KUKA KRL program: MyProgram_042().src

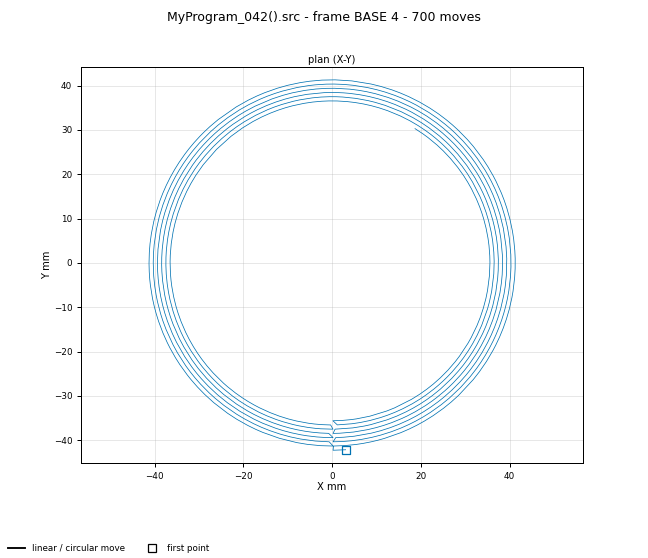
[picture p0: tool path of MyProgram_042().src in frame BASE 4, 700 of 700 moves have a stored position in this frame; points joined in program order, loops and branches not executed]
&ACCESS RVP
&REL 1
&PARAM TEMPLATE = C:\KRC\Roboter\Template\vorgabe
&PARAM EDITMASK = *
DEF MyProgram_042()
; ---- Setting reference (Base) ----
$BASE = BASE_DATA[4]

; --------------------------
; ---- Setting tool (TCP) ----
$TOOL = TOOL_DATA[3]
; --------------------------

$VEL.CP = VEL_APROX_PRINT
Startdeposition()
$VEL.CP = VEL_PRINT
LIN {X 3.0442,Y -42.1231,Z 63,A -93.24,B 24.8701,C -2.6301,E1 25.0087,E2 -183.3555} C_DIS
LIN {X 0.2102,Y -42.232,Z 63,A -95.217,B 24.8675,C -2.6563,E1 25.0033,E2 -181.4412} C_DIS
Enddeposition()
LIN {X 0.2102,Y -42.232,Z 63,A -95.217,B 24.8675,C -2.6563,E1 25.0033,E2 -181.4412} C_DIS
Startdeposition()
$VEL.CP = VEL_PRINT
LIN {X 0.315,Y -41.2814,Z 63,A -95.2944,B 24.8662,C -2.6692,E1 25.0033,E2 -181.3947} C_DIS
LIN {X 2.8307,Y -41.1855,Z 63,A -91.2878,B 24.8653,C -2.6781,E1 25.0144,E2 -185.421} C_DIS
LIN {X 5.3557,Y -40.9338,Z 63,A -88.2842,B 24.8659,C -2.6725,E1 25.0227,E2 -188.409} C_DIS
LIN {X 6.9926,Y -40.6865,Z 63,A -85.9418,B 24.8656,C -2.6748,E1 25.0292,E2 -190.7546} C_DIS
LIN {X 8.7788,Y -40.3384,Z 63,A -83.5592,B 24.8656,C -2.6748,E1 25.0357,E2 -193.1343} C_DIS
LIN {X 10.339,Y -39.9671,Z 63,A -81.3025,B 24.8654,C -2.6775,E1 25.0418,E2 -195.3939} C_DIS
LIN {X 11.8031,Y -39.5594,Z 63,A -78.4268,B 24.8639,C -2.6916,E1 25.0496,E2 -198.2983} C_DIS
LIN {X 15.4835,Y -38.2691,Z 63,A -73.5141,B 24.864,C -2.6909,E1 25.0624,E2 -203.1988} C_DIS
LIN {X 17.356,Y -37.457,Z 63,A -70.9592,B 24.864,C -2.6907,E1 25.0689,E2 -205.747} C_DIS
LIN {X 19.1269,Y -36.5846,Z 63,A -67.9342,B 24.8631,C -2.6997,E1 25.0765,E2 -208.785} C_DIS
LIN {X 20.771,Y -35.6773,Z 63,A -65.7267,B 24.8633,C -2.6979,E1 25.0818,E2 -210.9816} C_DIS
LIN {X 22.743,Y -34.453,Z 63,A -61.7056,B 24.8614,C -2.7169,E1 25.0913,E2 -215.0347} C_DIS
LIN {X 25.1016,Y -32.7747,Z 63,A -58.6078,B 24.8621,C -2.7101,E1 25.0982,E2 -218.1053} C_DIS
LIN {X 26.8177,Y -31.3859,Z 63,A -54.5171,B 24.8596,C -2.7337,E1 25.1071,E2 -222.2362} C_DIS
LIN {X 28.5068,Y -29.8606,Z 63,A -51.198,B 24.8586,C -2.7437,E1 25.1138,E2 -225.5653} C_DIS
LIN {X 31.826,Y -26.2941,Z 63,A -45.9801,B 24.8596,C -2.7345,E1 25.1235,E2 -230.7384} C_DIS
LIN {X 33.2022,Y -24.5336,Z 63,A -41.6673,B 24.8566,C -2.7631,E1 25.1308,E2 -235.0984} C_DIS
LIN {X 34.8038,Y -22.2027,Z 63,A -38.0776,B 24.8561,C -2.7682,E1 25.1363,E2 -238.682} C_DIS
LIN {X 36.2645,Y -19.7265,Z 63,A -34.6826,B 24.856,C -2.7693,E1 25.141,E2 -242.0622} C_DIS
LIN {X 36.8871,Y -18.5378,Z 63,A -32.5636,B 24.8549,C -2.7791,E1 25.1437,E2 -244.193} C_DIS
LIN {X 37.7579,Y -16.6921,Z 63,A -29.815,B 24.8542,C -2.786,E1 25.1469,E2 -246.9431} C_DIS
LIN {X 38.5649,Y -14.7316,Z 63,A -26.6228,B 24.8528,C -2.7991,E1 25.1502,E2 -250.1487} C_DIS
LIN {X 39.282,Y -12.6955,Z 63,A -23.7097,B 24.852,C -2.8068,E1 25.1528,E2 -253.0635} C_DIS
LIN {X 39.9316,Y -10.477,Z 63,A -20.4876,B 24.8509,C -2.8169,E1 25.1552,E2 -256.291} C_DIS
LIN {X 40.5343,Y -7.8247,Z 63,A -17.1592,B 24.8505,C -2.8209,E1 25.1571,E2 -259.6096} C_DIS
LIN {X 40.7866,Y -6.3807,Z 63,A -14.5033,B 24.8487,C -2.8381,E1 25.1583,E2 -262.2905} C_DIS
LIN {X 41.1553,Y -3.24,Z 63,A -10.513,B 24.8479,C -2.8449,E1 25.1594,E2 -266.2733} C_DIS
LIN {X 41.2627,Y -1.282,Z 63,A -7.9389,B 24.8473,C -2.8509,E1 25.1597,E2 -268.8463} C_DIS
LIN {X 41.2709,Y 1.0166,Z 63,A -4.6576,B 24.8461,C -2.8625,E1 25.1597,E2 -272.1355} C_DIS
LIN {X 41.1906,Y 2.7556,Z 63,A -2.0891,B 24.845,C -2.8727,E1 25.1592,E2 -274.7128} C_DIS
LIN {X 40.9304,Y 5.3819,Z 63,A 1.2618,B 24.8443,C -2.8786,E1 25.1582,E2 -278.0579} C_DIS
LIN {X 40.6503,Y 7.1984,Z 63,A 3.8015,B 24.8435,C -2.8862,E1 25.157,E2 -280.6007} C_DIS
LIN {X 40.085,Y 9.8718,Z 63,A 7.7678,B 24.8419,C -2.9006,E1 25.1546,E2 -284.5781} C_DIS
LIN {X 39.3831,Y 12.3781,Z 63,A 11.2245,B 24.841,C -2.9086,E1 25.1519,E2 -288.0339} C_DIS
LIN {X 38.8049,Y 14.0869,Z 63,A 13.9911,B 24.8397,C -2.9203,E1 25.1493,E2 -290.8127} C_DIS
LIN {X 38.1479,Y 15.7808,Z 63,A 16.574,B 24.8388,C -2.9285,E1 25.1465,E2 -293.4007} C_DIS
LIN {X 36.9226,Y 18.4657,Z 63,A 20.0406,B 24.8388,C -2.9291,E1 25.1424,E2 -296.85} C_DIS
LIN {X 36.2981,Y 19.6648,Z 63,A 22.4905,B 24.8372,C -2.9437,E1 25.1392,E2 -299.3218} C_DIS
LIN {X 35.1309,Y 21.6821,Z 63,A 25.3607,B 24.8369,C -2.946,E1 25.1351,E2 -302.1826} C_DIS
LIN {X 34.0764,Y 23.3033,Z 63,A 28.3406,B 24.8356,C -2.9576,E1 25.1304,E2 -305.1752} C_DIS
LIN {X 31.8607,Y 26.2512,Z 63,A 33.4994,B 24.8342,C -2.9703,E1 25.1215,E2 -310.3398} C_DIS
LIN {X 30.509,Y 27.8114,Z 63,A 36.4108,B 24.8334,C -2.9773,E1 25.1161,E2 -313.2549} C_DIS
LIN {X 28.3817,Y 29.9792,Z 63,A 40.0226,B 24.8335,C -2.9762,E1 25.1089,E2 -316.8489} C_DIS
LIN {X 27.0729,Y 31.1661,Z 63,A 42.6358,B 24.8327,C -2.9835,E1 25.1035,E2 -319.469} C_DIS
LIN {X 25.7131,Y 32.2973,Z 63,A 45.1305,B 24.8321,C -2.9886,E1 25.0981,E2 -321.9664} C_DIS
LIN {X 23.9669,Y 33.6129,Z 63,A 48.357,B 24.8312,C -2.9968,E1 25.0908,E2 -325.2008} C_DIS
LIN {X 22.0438,Y 34.9044,Z 63,A 51.6022,B 24.8306,C -3.0022,E1 25.0832,E2 -328.4482} C_DIS
LIN {X 19.7088,Y 36.2742,Z 63,A 55.2508,B 24.8302,C -3.0056,E1 25.0743,E2 -332.0942} C_DIS
LIN {X 17.2496,Y 37.5061,Z 63,A 58.8402,B 24.8301,C -3.0067,E1 25.0653,E2 -335.6767} C_DIS
LIN {X 15.2686,Y 38.3557,Z 63,A 61.9376,B 24.8296,C -3.0113,E1 25.0573,E2 -338.7779} C_DIS
LIN {X 13.4538,Y 39.0293,Z 63,A 64.4175,B 24.8296,C -3.0106,E1 25.0508,E2 -341.2509} C_DIS
LIN {X 11.0382,Y 39.7796,Z 63,A 68.6726,B 24.8281,C -3.024,E1 25.0393,E2 -345.5307} C_DIS
LIN {X 8.7687,Y 40.3406,Z 63,A 72.0577,B 24.8277,C -3.0276,E1 25.0301,E2 -348.9199} C_DIS
LIN {X 4.4531,Y 41.042,Z 63,A 77.9984,B 24.8277,C -3.0271,E1 25.0137,E2 -354.8545} C_DIS
LIN {X 0.6654,Y 41.2774,Z 63,A 82.6151,B 24.8288,C -3.0177,E1 25.0008,E2 -359.4473} C_DIS
LIN {X -2.2833,Y 41.2194,Z 63,A 87.1591,B 24.8283,C -3.0226,E1 24.9881,E2 -364.0039} C_DIS
LIN {X -5.0199,Y 40.9768,Z 63,A 90.6583,B 24.829,C -3.0164,E1 24.9784,E2 -367.4903} C_DIS
LIN {X -7.1609,Y 40.6571,Z 63,A 93.4772,B 24.8295,C -3.0118,E1 24.9707,E2 -370.3009} C_DIS
LIN {X -9.9422,Y 40.0677,Z 63,A 98.312,B 24.8286,C -3.02,E1 24.9575,E2 -375.1616} C_DIS
LIN {X -12.3271,Y 39.3993,Z 63,A 101.3903,B 24.8295,C -3.0115,E1 24.9493,E2 -378.225} C_DIS
LIN {X -15.2193,Y 38.3746,Z 63,A 105.1565,B 24.8309,C -2.9998,E1 24.9395,E2 -381.971} C_DIS
LIN {X -16.9866,Y 37.6259,Z 63,A 107.9518,B 24.8311,C -2.9977,E1 24.9324,E2 -384.7678} C_DIS
LIN {X -18.9393,Y 36.6822,Z 63,A 111.1263,B 24.8314,C -2.995,E1 24.9244,E2 -387.9443} C_DIS
LIN {X -21.6363,Y 35.1594,Z 63,A 116.2699,B 24.8311,C -2.9978,E1 24.912,E2 -393.1102} C_DIS
LIN {X -25.6799,Y 32.3235,Z 63,A 122.2724,B 24.8338,C -2.9736,E1 24.8986,E2 -399.0763} C_DIS
LIN {X -27.5314,Y 30.7617,Z 63,A 125.6343,B 24.8346,C -2.9662,E1 24.8916,E2 -402.4337} C_DIS
LIN {X -28.875,Y 29.5046,Z 63,A 127.9005,B 24.8357,C -2.957,E1 24.887,E2 -404.6872} C_DIS
LIN {X -29.8566,Y 28.5109,Z 63,A 129.8633,B 24.8362,C -2.9526,E1 24.8832,E2 -406.648} C_DIS
LIN {X -31.0997,Y 27.1489,Z 63,A 132.6919,B 24.8365,C -2.9494,E1 24.8779,E2 -409.4817} C_DIS
LIN {X -32.2803,Y 25.7346,Z 63,A 134.9712,B 24.8376,C -2.9397,E1 24.8739,E2 -411.7483} C_DIS
LIN {X -33.2684,Y 24.4433,Z 63,A 137.2968,B 24.8382,C -2.9346,E1 24.87,E2 -414.0728} C_DIS
LIN {X -34.5023,Y 22.6682,Z 63,A 140.7751,B 24.8385,C -2.9319,E1 24.8646,E2 -417.5619} C_DIS
LIN {X -35.5264,Y 21.0269,Z 63,A 143.1596,B 24.8397,C -2.921,E1 24.8612,E2 -419.9327} C_DIS
LIN {X -36.4931,Y 19.3006,Z 63,A 145.7888,B 24.8407,C -2.9119,E1 24.8577,E2 -422.5541} C_DIS
LIN {X -37.4028,Y 17.4725,Z 63,A 148.9048,B 24.8412,C -2.9068,E1 24.8539,E2 -425.6746} C_DIS
LIN {X -38.1649,Y 15.7395,Z 63,A 151.2341,B 24.8424,C -2.8957,E1 24.8514,E2 -427.9904} C_DIS
LIN {X -38.7933,Y 14.1186,Z 63,A 153.8854,B 24.8429,C -2.8911,E1 24.8488,E2 -430.6456} C_DIS
LIN {X -39.6647,Y 11.4457,Z 63,A 157.3648,B 24.8447,C -2.8746,E1 24.8459,E2 -434.1055} C_DIS
LIN {X -40.2119,Y 9.3412,Z 63,A 161.2523,B 24.8447,C -2.8748,E1 24.8432,E2 -438.0161} C_DIS
LIN {X -40.7666,Y 6.5072,Z 63,A 165.1234,B 24.8462,C -2.8608,E1 24.8414,E2 -441.8767} C_DIS
LIN {X -41.0514,Y 4.3638,Z 63,A 167.693,B 24.8478,C -2.8467,E1 24.8405,E2 -444.4279} C_DIS
LIN {X -41.2148,Y 2.3664,Z 63,A 170.8387,B 24.8483,C -2.8419,E1 24.8399,E2 -447.5811} C_DIS
LIN {X -41.2825,Y -0.1257,Z 63,A 173.8276,B 24.85,C -2.826,E1 24.8398,E2 -450.5498} C_DIS
LIN {X -41.2319,Y -2.0447,Z 63,A 176.7215,B 24.8506,C -2.8201,E1 24.8401,E2 -453.4472} C_DIS
LIN {X -41.1157,Y -3.7096,Z 63,A 178.9624,B 24.8514,C -2.8121,E1 24.8406,E2 -455.6824} C_DIS
LIN {X -40.9765,Y -5.0234,Z 63,A -178.6298,B 24.8514,C -2.8128,E1 24.8414,E2 -458.1061} C_DIS
LIN {X -40.4873,Y -8.0658,Z 63,A -174.7424,B 24.8532,C -2.7954,E1 24.8432,E2 -461.9751} C_DIS
LIN {X -40.0866,Y -9.8654,Z 63,A -172.1473,B 24.854,C -2.7882,E1 24.8449,E2 -464.568} C_DIS
LIN {X -39.674,Y -11.413,Z 63,A -170.0611,B 24.8548,C -2.7801,E1 24.8464,E2 -466.6469} C_DIS
LIN {X -39.1144,Y -13.2029,Z 63,A -167.1196,B 24.8552,C -2.7763,E1 24.849,E2 -469.5962} C_DIS
LIN {X -38.1488,Y -15.7789,Z 63,A -163.1877,B 24.8562,C -2.7667,E1 24.853,E2 -473.5272} C_DIS
LIN {X -37.1675,Y -17.9678,Z 63,A -160.3099,B 24.8577,C -2.7524,E1 24.8564,E2 -476.3866} C_DIS
LIN {X -36.5638,Y -19.1664,Z 63,A -158.0107,B 24.8577,C -2.7524,E1 24.8593,E2 -478.6981} C_DIS
LIN {X -35.3355,Y -21.3457,Z 63,A -154.537,B 24.8586,C -2.7434,E1 24.8642,E2 -482.1684} C_DIS
LIN {X -34.341,Y -22.9129,Z 63,A -151.7472,B 24.859,C -2.7395,E1 24.8685,E2 -484.9627} C_DIS
LIN {X -32.6576,Y -25.2536,Z 63,A -148.3403,B 24.8607,C -2.723,E1 24.8741,E2 -488.3465} C_DIS
LIN {X -31.8669,Y -26.2441,Z 63,A -146.1604,B 24.8607,C -2.7239,E1 24.878,E2 -490.5388} C_DIS
LIN {X -30.3612,Y -27.9725,Z 63,A -143.0206,B 24.8614,C -2.7164,E1 24.8838,E2 -493.6748} C_DIS
LIN {X -28.7127,Y -29.6617,Z 63,A -139.6987,B 24.862,C -2.7103,E1 24.8904,E2 -496.996} C_DIS
LIN {X -26.6654,Y -31.5156,Z 63,A -135.2889,B 24.862,C -2.7101,E1 24.8997,E2 -501.4227} C_DIS
LIN {X -23.5731,Y -33.8905,Z 63,A -130.0918,B 24.8633,C -2.6983,E1 24.9114,E2 -506.6101} C_DIS
LIN {X -21.5024,Y -35.2407,Z 63,A -126.7529,B 24.8639,C -2.6921,E1 24.9193,E2 -509.9447} C_DIS
LIN {X -19.0548,Y -36.6218,Z 63,A -123.185,B 24.8648,C -2.6828,E1 24.928,E2 -513.5004} C_DIS
LIN {X -17.1898,Y -37.5339,Z 63,A -120.338,B 24.8652,C -2.679,E1 24.9352,E2 -516.3457} C_DIS
LIN {X -15.6398,Y -38.2055,Z 63,A -117.3395,B 24.8646,C -2.6854,E1 24.943,E2 -519.3661} C_DIS
LIN {X -11.9039,Y -39.5295,Z 63,A -111.6303,B 24.8647,C -2.684,E1 24.9581,E2 -525.0825} C_DIS
LIN {X -7.9714,Y -40.5061,Z 63,A -107.0486,B 24.8664,C -2.6669,E1 24.9705,E2 -529.6295} C_DIS
LIN {X -5.6211,Y -40.8983,Z 63,A -102.6413,B 24.865,C -2.6816,E1 24.9828,E2 -534.0754} C_DIS
LIN {X -2.6104,Y -41.2002,Z 63,A -98.9251,B 24.8657,C -2.6746,E1 24.9931,E2 -537.7766} C_DIS
LIN {X 0.2191,Y -41.2805,Z 63,A -96.8151,B 24.8682,C -2.6493,E1 24.9988,E2 -539.8267} C_DIS
Enddeposition()
LIN {X 0.2191,Y -41.2805,Z 63,A -96.8151,B 24.8682,C -2.6493,E1 24.9988,E2 -539.8267} C_DIS
Startdeposition()
$VEL.CP = VEL_PRINT
LIN {X -0.6723,Y -40.3269,Z 63,A -98.638,B 24.8673,C -2.6582,E1 24.9938,E2 -538.0247} C_DIS
LIN {X -3.7987,Y -40.1536,Z 63,A -102.8793,B 24.867,C -2.661,E1 24.982,E2 -533.7884} C_DIS
LIN {X -7.1068,Y -39.7017,Z 63,A -106.8696,B 24.8659,C -2.6722,E1 24.971,E2 -529.8212} C_DIS
LIN {X -9.4207,Y -39.2174,Z 63,A -111.0995,B 24.8669,C -2.6624,E1 24.9594,E2 -525.5625} C_DIS
LIN {X -11.7387,Y -38.5874,Z 63,A -114.2382,B 24.8663,C -2.6681,E1 24.9511,E2 -522.4324} C_DIS
LIN {X -14.0146,Y -37.82,Z 63,A -117.3497,B 24.8657,C -2.6747,E1 24.9429,E2 -519.3306} C_DIS
LIN {X -15.9354,Y -37.0518,Z 63,A -120.4596,B 24.8656,C -2.6755,E1 24.9348,E2 -516.2155} C_DIS
LIN {X -17.6856,Y -36.2491,Z 63,A -122.93,B 24.8649,C -2.6819,E1 24.9286,E2 -513.754} C_DIS
LIN {X -19.7095,Y -35.1891,Z 63,A -126.7906,B 24.8653,C -2.6786,E1 24.9191,E2 -509.8748} C_DIS
LIN {X -21.525,Y -34.1093,Z 63,A -129.8482,B 24.8649,C -2.6824,E1 24.9119,E2 -506.8163} C_DIS
LIN {X -24.3338,Y -32.1655,Z 63,A -134.5954,B 24.8639,C -2.6916,E1 24.9011,E2 -502.0747} C_DIS
LIN {X -26.3607,Y -30.5267,Z 63,A -138.0135,B 24.8629,C -2.7017,E1 24.8938,E2 -498.6676} C_DIS
LIN {X -27.723,Y -29.2947,Z 63,A -140.8695,B 24.8627,C -2.7041,E1 24.888,E2 -495.8055} C_DIS
LIN {X -29.6846,Y -27.305,Z 63,A -144.4563,B 24.8614,C -2.7168,E1 24.8811,E2 -492.2336} C_DIS
LIN {X -30.9078,Y -25.9128,Z 63,A -147.0794,B 24.8608,C -2.7227,E1 24.8763,E2 -489.6128} C_DIS
LIN {X -31.9763,Y -24.5815,Z 63,A -149.52,B 24.8602,C -2.7282,E1 24.8721,E2 -487.1738} C_DIS
LIN {X -32.9916,Y -23.2011,Z 63,A -152.5473,B 24.8602,C -2.7276,E1 24.8672,E2 -484.1302} C_DIS
LIN {X -34.8756,Y -20.2598,Z 63,A -157.4876,B 24.8589,C -2.7405,E1 24.86,E2 -479.1955} C_DIS
LIN {X -35.8631,Y -18.4549,Z 63,A -160.6337,B 24.8584,C -2.746,E1 24.8559,E2 -476.0457} C_DIS
LIN {X -37.4233,Y -15.0421,Z 63,A -165.3478,B 24.8562,C -2.7673,E1 24.8507,E2 -471.3567} C_DIS
LIN {X -38.1586,Y -13.0647,Z 63,A -168.5623,B 24.8555,C -2.7737,E1 24.8477,E2 -468.1391} C_DIS
LIN {X -38.6645,Y -11.48,Z 63,A -171.1673,B 24.855,C -2.7781,E1 24.8456,E2 -465.5297} C_DIS
LIN {X -39.3705,Y -8.7591,Z 63,A -174.6366,B 24.8532,C -2.7955,E1 24.8433,E2 -462.0816} C_DIS
LIN {X -39.6731,Y -7.2657,Z 63,A -177.011,B 24.8527,C -2.7999,E1 24.8421,E2 -459.7037} C_DIS
LIN {X -39.9923,Y -5.2302,Z 63,A -179.865,B 24.8517,C -2.8096,E1 24.8409,E2 -456.856} C_DIS
LIN {X -40.2241,Y -2.9686,Z 63,A 176.0361,B 24.8516,C -2.8108,E1 24.84,E2 -452.7352} C_DIS
LIN {X -40.3332,Y 0.0142,Z 63,A 172.5148,B 24.8494,C -2.8313,E1 24.8398,E2 -449.2418} C_DIS
LIN {X -40.279,Y 2.0829,Z 63,A 169.4008,B 24.8486,C -2.8388,E1 24.8401,E2 -446.1269} C_DIS
LIN {X -40.1128,Y 4.2063,Z 63,A 165.9993,B 24.848,C -2.8445,E1 24.8411,E2 -442.7187} C_DIS
LIN {X -39.6244,Y 7.5267,Z 63,A 161.4804,B 24.8461,C -2.8618,E1 24.8431,E2 -438.2145} C_DIS
LIN {X -38.9796,Y 10.3609,Z 63,A 157.4198,B 24.8447,C -2.8753,E1 24.8458,E2 -434.1624} C_DIS
LIN {X -38.1564,Y 13.0713,Z 63,A 153.0309,B 24.8437,C -2.8838,E1 24.8496,E2 -429.7687} C_DIS
LIN {X -37.1679,Y 15.6614,Z 63,A 149.2433,B 24.8423,C -2.8971,E1 24.8535,E2 -425.9918} C_DIS
LIN {X -36.2263,Y 17.7322,Z 63,A 146.4377,B 24.8408,C -2.9109,E1 24.8569,E2 -423.204} C_DIS
LIN {X -35.3698,Y 19.384,Z 63,A 143.596,B 24.8402,C -2.9164,E1 24.8606,E2 -420.3603} C_DIS
LIN {X -34.4492,Y 20.9759,Z 63,A 141.2131,B 24.8391,C -2.9261,E1 24.864,E2 -417.9884} C_DIS
LIN {X -33.4645,Y 22.5138,Z 63,A 138.3387,B 24.8387,C -2.9302,E1 24.8684,E2 -415.1093} C_DIS
LIN {X -32.4432,Y 23.9625,Z 63,A 136.0696,B 24.8376,C -2.9395,E1 24.8721,E2 -412.8515} C_DIS
LIN {X -31.4476,Y 25.255,Z 63,A 133.6511,B 24.8371,C -2.9444,E1 24.8762,E2 -410.4333} C_DIS
LIN {X -29.9352,Y 27.0299,Z 63,A 129.6912,B 24.8369,C -2.9457,E1 24.8836,E2 -406.4586} C_DIS
LIN {X -27.4236,Y 29.5748,Z 63,A 124.7893,B 24.8354,C -2.9594,E1 24.8933,E2 -401.569} C_DIS
LIN {X -25.668,Y 31.1112,Z 63,A 121.871,B 24.8341,C -2.971,E1 24.8995,E2 -398.6672} C_DIS
LIN {X -23.5027,Y 32.7775,Z 63,A 117.1805,B 24.8342,C -2.9698,E1 24.9101,E2 -393.957} C_DIS
LIN {X -20.9052,Y 34.4921,Z 63,A 113.3733,B 24.8325,C -2.9849,E1 24.919,E2 -390.1739} C_DIS
LIN {X -18.8345,Y 35.6651,Z 63,A 109.6522,B 24.8324,C -2.9866,E1 24.9281,E2 -386.4462} C_DIS
LIN {X -16.3132,Y 36.8866,Z 63,A 106.4728,B 24.8306,C -3.0021,E1 24.9361,E2 -383.2956} C_DIS
LIN {X -14.6293,Y 37.5863,Z 63,A 103.5697,B 24.8306,C -3.0018,E1 24.9436,E2 -380.3855} C_DIS
LIN {X -12.9467,Y 38.1984,Z 63,A 100.8236,B 24.8306,C -3.0025,E1 24.9509,E2 -377.6356} C_DIS
LIN {X -11.1981,Y 38.747,Z 63,A 97.7211,B 24.8309,C -2.9992,E1 24.9592,E2 -374.5202} C_DIS
LIN {X -7.9066,Y 39.5508,Z 63,A 93.2503,B 24.83,C -3.0076,E1 24.9714,E2 -370.0637} C_DIS
LIN {X -5.2768,Y 39.986,Z 63,A 89.8662,B 24.8291,C -3.0152,E1 24.9807,E2 -366.6949} C_DIS
LIN {X -3.7844,Y 40.1549,Z 63,A 87.3873,B 24.8295,C -3.0119,E1 24.9876,E2 -364.2066} C_DIS
LIN {X -1.3223,Y 40.311,Z 63,A 83.8807,B 24.8294,C -3.0131,E1 24.9973,E2 -360.7019} C_DIS
LIN {X 0.4163,Y 40.331,Z 63,A 81.3218,B 24.8294,C -3.0124,E1 25.0045,E2 -358.1415} C_DIS
LIN {X 2.6441,Y 40.2461,Z 63,A 78.4388,B 24.829,C -3.0162,E1 25.0125,E2 -355.2687} C_DIS
LIN {X 4.7439,Y 40.0529,Z 63,A 74.9846,B 24.8297,C -3.0096,E1 25.0221,E2 -351.8012} C_DIS
LIN {X 7.9549,Y 39.5409,Z 63,A 70.9226,B 24.8291,C -3.0157,E1 25.0332,E2 -347.7578} C_DIS
LIN {X 10.1713,Y 39.0292,Z 63,A 67.5872,B 24.8294,C -3.0125,E1 25.0423,E2 -344.4196} C_DIS
LIN {X 11.9463,Y 38.523,Z 63,A 64.861,B 24.8298,C -3.0091,E1 25.0496,E2 -341.6903} C_DIS
LIN {X 14.0403,Y 37.8106,Z 63,A 61.8691,B 24.8298,C -3.0086,E1 25.0575,E2 -338.703} C_DIS
LIN {X 15.6139,Y 37.1879,Z 63,A 59.3682,B 24.8303,C -3.0048,E1 25.0639,E2 -336.1988} C_DIS
LIN {X 17.4857,Y 36.3454,Z 63,A 56.573,B 24.8305,C -3.0032,E1 25.071,E2 -333.4071} C_DIS
LIN {X 19.0006,Y 35.5773,Z 63,A 53.6808,B 24.8316,C -2.9931,E1 25.0782,E2 -330.4989} C_DIS
LIN {X 21.8543,Y 33.8988,Z 63,A 49.8608,B 24.8309,C -2.9994,E1 25.0873,E2 -326.7058} C_DIS
LIN {X 23.7603,Y 32.5912,Z 63,A 45.7015,B 24.833,C -2.9808,E1 25.0968,E2 -322.5168} C_DIS
LIN {X 25.5002,Y 31.2489,Z 63,A 43.1956,B 24.8326,C -2.9846,E1 25.1023,E2 -320.0291} C_DIS
LIN {X 26.5953,Y 30.3222,Z 63,A 41.107,B 24.8331,C -2.9799,E1 25.1067,E2 -317.9377} C_DIS
LIN {X 27.705,Y 29.3117,Z 63,A 38.678,B 24.8341,C -2.9711,E1 25.1117,E2 -315.4977} C_DIS
LIN {X 29.529,Y 27.4728,Z 63,A 35.2524,B 24.8345,C -2.9673,E1 25.1183,E2 -312.0778} C_DIS
LIN {X 31.1134,Y 25.6654,Z 63,A 31.3937,B 24.8362,C -2.9526,E1 25.1253,E2 -308.2019} C_DIS
LIN {X 32.6965,Y 23.6163,Z 63,A 27.6778,B 24.8372,C -2.9432,E1 25.1315,E2 -304.4816} C_DIS
LIN {X 34.4358,Y 20.998,Z 63,A 23.9494,B 24.8372,C -2.9437,E1 25.1371,E2 -300.7731} C_DIS
LIN {X 35.1373,Y 19.8015,Z 63,A 21.9628,B 24.8378,C -2.9383,E1 25.1399,E2 -298.7839} C_DIS
LIN {X 35.8718,Y 18.4379,Z 63,A 19.7335,B 24.8385,C -2.9319,E1 25.1428,E2 -296.5513} C_DIS
LIN {X 36.7127,Y 16.7012,Z 63,A 16.6795,B 24.8399,C -2.9193,E1 25.1464,E2 -293.4839} C_DIS
LIN {X 37.4691,Y 14.9279,Z 63,A 14.2702,B 24.8401,C -2.917,E1 25.149,E2 -291.0823} C_DIS
LIN {X 38.2617,Y 12.759,Z 63,A 10.3402,B 24.8423,C -2.8969,E1 25.1526,E2 -287.1268} C_DIS
LIN {X 38.9421,Y 10.4999,Z 63,A 7.5435,B 24.8424,C -2.896,E1 25.1548,E2 -284.3442} C_DIS
LIN {X 39.5395,Y 7.9614,Z 63,A 3.4265,B 24.8444,C -2.8781,E1 25.1572,E2 -280.2087} C_DIS
LIN {X 39.942,Y 5.6015,Z 63,A -0.1327,B 24.8458,C -2.865,E1 25.1587,E2 -276.6395} C_DIS
LIN {X 40.2893,Y 1.8711,Z 63,A -4.9516,B 24.8467,C -2.8568,E1 25.1597,E2 -271.8298} C_DIS
LIN {X 40.3236,Y -0.8722,Z 63,A -9.1136,B 24.8485,C -2.8402,E1 25.1597,E2 -267.6533} C_DIS
LIN {X 40.2198,Y -3.0229,Z 63,A -12.1864,B 24.8495,C -2.8304,E1 25.1591,E2 -264.5753} C_DIS
LIN {X 39.8473,Y -6.2392,Z 63,A -16.2724,B 24.8501,C -2.8245,E1 25.1576,E2 -260.4995} C_DIS
LIN {X 39.5044,Y -8.1325,Z 63,A -18.9712,B 24.851,C -2.8165,E1 25.1561,E2 -257.7978} C_DIS
LIN {X 39.1186,Y -9.8242,Z 63,A -21.3873,B 24.8517,C -2.8097,E1 25.1546,E2 -255.3794} C_DIS
LIN {X 38.7142,Y -11.3126,Z 63,A -23.4528,B 24.8522,C -2.805,E1 25.153,E2 -253.3148} C_DIS
LIN {X 38.2315,Y -12.8487,Z 63,A -25.8167,B 24.8531,C -2.7968,E1 25.151,E2 -250.9447} C_DIS
LIN {X 37.5984,Y -14.5986,Z 63,A -28.5362,B 24.854,C -2.7876,E1 25.1483,E2 -248.2186} C_DIS
LIN {X 36.9237,Y -16.2293,Z 63,A -30.9038,B 24.8546,C -2.7824,E1 25.1457,E2 -245.8518} C_DIS
LIN {X 36.2858,Y -17.6097,Z 63,A -32.9712,B 24.8551,C -2.7776,E1 25.1432,E2 -243.7842} C_DIS
LIN {X 35.5224,Y -19.1027,Z 63,A -35.5389,B 24.8561,C -2.7677,E1 25.1399,E2 -241.2065} C_DIS
LIN {X 34.5887,Y -20.7464,Z 63,A -38.1715,B 24.8568,C -2.761,E1 25.1362,E2 -238.5716} C_DIS
LIN {X 33.5695,Y -22.3575,Z 63,A -40.9006,B 24.8576,C -2.7532,E1 25.132,E2 -235.8378} C_DIS
LIN {X 32.5771,Y -23.7795,Z 63,A -43.1766,B 24.858,C -2.7496,E1 25.1283,E2 -233.5644} C_DIS
LIN {X 31.1406,Y -25.6326,Z 63,A -46.8133,B 24.8594,C -2.736,E1 25.122,E2 -229.9125} C_DIS
LIN {X 28.9609,Y -28.0705,Z 63,A -51.7845,B 24.8611,C -2.7195,E1 25.1125,E2 -224.9239} C_DIS
LIN {X 26.4435,Y -30.4544,Z 63,A -56.8908,B 24.8625,C -2.7055,E1 25.1019,E2 -219.8049} C_DIS
LIN {X 24.6004,Y -31.9618,Z 63,A -59.5165,B 24.8621,C -2.7101,E1 25.0962,E2 -217.2} C_DIS
LIN {X 22.1544,Y -33.7034,Z 63,A -63.5632,B 24.8626,C -2.7051,E1 25.087,E2 -213.1552} C_DIS
LIN {X 20.532,Y -34.7155,Z 63,A -66.5739,B 24.8635,C -2.6956,E1 25.0797,E2 -210.1314} C_DIS
LIN {X 18.9264,Y -35.6167,Z 63,A -68.934,B 24.8636,C -2.695,E1 25.074,E2 -207.7769} C_DIS
LIN {X 17.294,Y -36.4375,Z 63,A -71.7425,B 24.8643,C -2.6877,E1 25.0669,E2 -204.9584} C_DIS
LIN {X 15.5479,Y -37.2158,Z 63,A -74.2772,B 24.8645,C -2.6865,E1 25.0604,E2 -202.4269} C_DIS
LIN {X 13.3753,Y -38.0504,Z 63,A -77.9999,B 24.8655,C -2.676,E1 25.0506,E2 -198.6872} C_DIS
LIN {X 10.9144,Y -38.828,Z 63,A -81.5928,B 24.8658,C -2.673,E1 25.041,E2 -195.0934} C_DIS
LIN {X 8.9724,Y -39.3223,Z 63,A -84.0709,B 24.8656,C -2.6756,E1 25.0343,E2 -192.6251} C_DIS
LIN {X 6.643,Y -39.782,Z 63,A -87.891,B 24.8665,C -2.6665,E1 25.0238,E2 -188.7877} C_DIS
LIN {X 4.3725,Y -40.0954,Z 63,A -90.7016,B 24.866,C -2.6708,E1 25.016,E2 -185.9895} C_DIS
LIN {X 2.215,Y -40.2719,Z 63,A -94.0044,B 24.8665,C -2.6663,E1 25.0068,E2 -182.6774} C_DIS
LIN {X 0.2157,Y -40.3237,Z 63,A -96.1344,B 24.8656,C -2.6755,E1 25.0009,E2 -180.5697} C_DIS
Enddeposition()
LIN {X 0.2157,Y -40.3237,Z 63,A -96.1344,B 24.8656,C -2.6755,E1 25.0009,E2 -180.5697} C_DIS
Startdeposition()
$VEL.CP = VEL_PRINT
LIN {X 0.8258,Y -39.3744,Z 63,A -94.5482,B 24.8629,C -2.7016,E1 25.0055,E2 -182.2178} C_DIS
LIN {X 2.6074,Y -39.2964,Z 63,A -91.716,B 24.8625,C -2.706,E1 25.0134,E2 -185.0593} C_DIS
LIN {X 5.0033,Y -39.0639,Z 63,A -87.8195,B 24.8617,C -2.7137,E1 25.0243,E2 -188.9711} C_DIS
LIN {X 8.8554,Y -38.3745,Z 63,A -82.9368,B 24.8624,C -2.7067,E1 25.0376,E2 -193.8314} C_DIS
LIN {X 10.9631,Y -37.8262,Z 63,A -79.3267,B 24.8614,C -2.7164,E1 25.0473,E2 -197.4589} C_DIS
LIN {X 13.1476,Y -37.1237,Z 63,A -76.1917,B 24.8614,C -2.7175,E1 25.0556,E2 -200.5903} C_DIS
LIN {X 15.0969,Y -36.3751,Z 63,A -73.1585,B 24.8609,C -2.7216,E1 25.0635,E2 -203.6264} C_DIS
LIN {X 17.1903,Y -35.4334,Z 63,A -69.5052,B 24.8599,C -2.7315,E1 25.0728,E2 -207.2937} C_DIS
LIN {X 18.903,Y -34.5501,Z 63,A -67.0771,B 24.8599,C -2.7305,E1 25.0787,E2 -209.7126} C_DIS
LIN {X 20.6091,Y -33.5604,Z 63,A -64.2704,B 24.8595,C -2.7347,E1 25.0855,E2 -212.5205} C_DIS
LIN {X 22.243,Y -32.5008,Z 63,A -61.2677,B 24.8587,C -2.7428,E1 25.0924,E2 -215.5324} C_DIS
LIN {X 23.9066,Y -31.297,Z 63,A -58.5206,B 24.8585,C -2.7452,E1 25.0986,E2 -218.2753} C_DIS
LIN {X 25.1491,Y -30.3074,Z 63,A -55.9218,B 24.8575,C -2.7547,E1 25.1042,E2 -220.8868} C_DIS
LIN {X 27.0288,Y -28.6437,Z 63,A -52.2888,B 24.8566,C -2.7627,E1 25.1117,E2 -224.5241} C_DIS
LIN {X 28.8769,Y -26.7793,Z 63,A -48.8811,B 24.8564,C -2.7653,E1 25.1183,E2 -227.9234} C_DIS
LIN {X 30.1971,Y -25.2819,Z 63,A -46.2276,B 24.856,C -2.7686,E1 25.1232,E2 -230.5727} C_DIS
LIN {X 31.1854,Y -24.0518,Z 63,A -43.4277,B 24.8545,C -2.7827,E1 25.128,E2 -233.3928} C_DIS
LIN {X 32.4975,Y -22.2468,Z 63,A -39.8312,B 24.853,C -2.7972,E1 25.1338,E2 -237.006} C_DIS
LIN {X 33.8363,Y -20.1516,Z 63,A -36.4821,B 24.8524,C -2.8029,E1 25.1387,E2 -240.3516} C_DIS
LIN {X 35.0666,Y -17.9263,Z 63,A -33.1056,B 24.8519,C -2.8082,E1 25.1431,E2 -243.7228} C_DIS
LIN {X 35.8645,Y -16.2717,Z 63,A -30.2453,B 24.8507,C -2.8191,E1 25.1465,E2 -246.5935} C_DIS
LIN {X 36.615,Y -14.5041,Z 63,A -27.7944,B 24.8504,C -2.8218,E1 25.1491,E2 -249.0373} C_DIS
LIN {X 37.3035,Y -12.628,Z 63,A -24.3708,B 24.8486,C -2.8392,E1 25.1523,E2 -252.4827} C_DIS
LIN {X 38.0133,Y -10.2946,Z 63,A -20.6352,B 24.8471,C -2.8532,E1 25.1552,E2 -256.2302} C_DIS
LIN {X 38.7596,Y -6.979,Z 63,A -16.4003,B 24.8467,C -2.8567,E1 25.1575,E2 -260.4488} C_DIS
LIN {X 39.022,Y -5.3238,Z 63,A -13.5925,B 24.8452,C -2.8705,E1 25.1587,E2 -263.2727} C_DIS
LIN {X 39.2819,Y -2.8243,Z 63,A -9.6627,B 24.8434,C -2.8866,E1 25.1596,E2 -267.2172} C_DIS
LIN {X 39.3715,Y 0.9706,Z 63,A -5.0597,B 24.8432,C -2.8886,E1 25.1597,E2 -271.7974} C_DIS
LIN {X 39.2108,Y 3.6786,Z 63,A 0.0271,B 24.8398,C -2.9198,E1 25.1586,E2 -276.9281} C_DIS
LIN {X 38.6024,Y 7.8031,Z 63,A 6.034,B 24.8379,C -2.9373,E1 25.1557,E2 -282.9411} C_DIS
LIN {X 37.8507,Y 10.8796,Z 63,A 10.1347,B 24.8373,C -2.9426,E1 25.1527,E2 -287.0308} C_DIS
LIN {X 36.9807,Y 13.5443,Z 63,A 13.84,B 24.8366,C -2.9483,E1 25.1494,E2 -290.7287} C_DIS
LIN {X 36.2362,Y 15.4265,Z 63,A 16.7113,B 24.8359,C -2.9554,E1 25.1463,E2 -293.6009} C_DIS
LIN {X 35.4954,Y 17.0612,Z 63,A 19.231,B 24.8352,C -2.9611,E1 25.1433,E2 -296.1205} C_DIS
LIN {X 34.5566,Y 18.8911,Z 63,A 22.3066,B 24.8342,C -2.9704,E1 25.1393,E2 -299.2021} C_DIS
LIN {X 33.7403,Y 20.3135,Z 63,A 24.9116,B 24.8331,C -2.9801,E1 25.1356,E2 -301.8167} C_DIS
LIN {X 32.3146,Y 22.5113,Z 63,A 28.726,B 24.832,C -2.9897,E1 25.1297,E2 -305.6348} C_DIS
LIN {X 31.2829,Y 23.9253,Z 63,A 31.3778,B 24.8311,C -2.9974,E1 25.1252,E2 -308.2922} C_DIS
LIN {X 29.4974,Y 26.0955,Z 63,A 34.949,B 24.8311,C -2.9985,E1 25.1187,E2 -311.8498} C_DIS
LIN {X 28.5457,Y 27.1331,Z 63,A 37.1973,B 24.8302,C -3.006,E1 25.1144,E2 -314.106} C_DIS
LIN {X 27.0284,Y 28.6442,Z 63,A 40.3953,B 24.8293,C -3.0136,E1 25.108,E2 -317.3088} C_DIS
LIN {X 25.0281,Y 30.4078,Z 63,A 44.0322,B 24.8289,C -3.0172,E1 25.1003,E2 -320.9401} C_DIS
LIN {X 23.458,Y 31.6353,Z 63,A 47.1054,B 24.828,C -3.0249,E1 25.0935,E2 -324.0202} C_DIS
LIN {X 21.4123,Y 33.0539,Z 63,A 50.8608,B 24.8271,C -3.0326,E1 25.0847,E2 -327.7814} C_DIS
LIN {X 19.462,Y 34.2375,Z 63,A 54.1315,B 24.8267,C -3.0366,E1 25.0769,E2 -331.0516} C_DIS
LIN {X 17.7248,Y 35.1696,Z 63,A 57.2095,B 24.8259,C -3.0432,E1 25.0692,E2 -334.137} C_DIS
LIN {X 14.8786,Y 36.4643,Z 63,A 61.3875,B 24.8259,C -3.0427,E1 25.0585,E2 -338.3036} C_DIS
LIN {X 12.6379,Y 37.3002,Z 63,A 65.1678,B 24.8251,C -3.05,E1 25.0485,E2 -342.0936} C_DIS
LIN {X 9.7365,Y 38.1605,Z 63,A 69.3775,B 24.8251,C -3.0501,E1 25.0372,E2 -346.2967} C_DIS
LIN {X 7.8233,Y 38.5982,Z 63,A 71.8161,B 24.8256,C -3.0457,E1 25.0306,E2 -348.7217} C_DIS
LIN {X 6.0046,Y 38.9225,Z 63,A 74.7769,B 24.8251,C -3.0503,E1 25.0224,E2 -351.6903} C_DIS
LIN {X 3.9713,Y 39.1824,Z 63,A 77.8908,B 24.8248,C -3.0525,E1 25.0138,E2 -354.8074} C_DIS
LIN {X 0.5943,Y 39.3787,Z 63,A 82.537,B 24.8253,C -3.0486,E1 25.0009,E2 -359.4428} C_DIS
LIN {X -1.3235,Y 39.3609,Z 63,A 85.4243,B 24.8253,C -3.0491,E1 24.9928,E2 -362.3317} C_DIS
LIN {X -3.6077,Y 39.2174,Z 63,A 88.6036,B 24.8256,C -3.0458,E1 24.984,E2 -365.5042} C_DIS
LIN {X -6.1695,Y 38.8965,Z 63,A 92.9067,B 24.8251,C -3.0504,E1 24.972,E2 -369.8218} C_DIS
LIN {X -8.9972,Y 38.3417,Z 63,A 97.0412,B 24.8256,C -3.0461,E1 24.9607,E2 -373.951} C_DIS
LIN {X -11.0798,Y 37.7925,Z 63,A 99.6437,B 24.8267,C -3.0363,E1 24.9538,E2 -376.5345} C_DIS
LIN {X -13.6028,Y 36.9594,Z 63,A 104.5969,B 24.8257,C -3.0448,E1 24.9407,E2 -381.5176} C_DIS
LIN {X -17.4048,Y 35.3284,Z 63,A 110.2096,B 24.8273,C -3.0311,E1 24.9265,E2 -387.1112} C_DIS
LIN {X -19.52,Y 34.2053,Z 63,A 113.1223,B 24.8287,C -3.0185,E1 24.9194,E2 -390.0024} C_DIS
LIN {X -21.2045,Y 33.1872,Z 63,A 116.2213,B 24.829,C -3.0161,E1 24.9121,E2 -393.1052} C_DIS
LIN {X -23.2441,Y 31.792,Z 63,A 120.0479,B 24.8295,C -3.0116,E1 24.9033,E2 -396.9343} C_DIS
LIN {X -25.1521,Y 30.305,Z 63,A 123.3632,B 24.8306,C -3.0019,E1 24.8961,E2 -400.2389} C_DIS
LIN {X -26.5449,Y 29.0929,Z 63,A 125.8445,B 24.8316,C -2.9936,E1 24.891,E2 -402.7103} C_DIS
LIN {X -27.5887,Y 28.1051,Z 63,A 127.8739,B 24.8322,C -2.9881,E1 24.8869,E2 -404.735} C_DIS
LIN {X -28.9944,Y 26.6522,Z 63,A 130.8497,B 24.8329,C -2.9814,E1 24.8812,E2 -407.7076} C_DIS
LIN {X -29.9606,Y 25.5613,Z 63,A 133.2476,B 24.8332,C -2.9791,E1 24.8768,E2 -410.111} C_DIS
LIN {X -31.3436,Y 23.8464,Z 63,A 136.4083,B 24.8342,C -2.9704,E1 24.8714,E2 -413.2656} C_DIS
LIN {X -32.385,Y 22.4107,Z 63,A 138.8083,B 24.8352,C -2.9616,E1 24.8675,E2 -415.6564} C_DIS
LIN {X -33.47,Y 20.7555,Z 63,A 142.1345,B 24.8355,C -2.9584,E1 24.8625,E2 -418.9918} C_DIS
LIN {X -34.7097,Y 18.6085,Z 63,A 145.7298,B 24.8367,C -2.9481,E1 24.8576,E2 -422.5813} C_DIS
LIN {X -35.8099,Y 16.3925,Z 63,A 149.4706,B 24.8377,C -2.9391,E1 24.8532,E2 -426.3208} C_DIS
LIN {X -36.7007,Y 14.2848,Z 63,A 152.9508,B 24.8386,C -2.9307,E1 24.8496,E2 -429.8005} C_DIS
LIN {X -37.7166,Y 11.3356,Z 63,A 157.0261,B 24.8406,C -2.9122,E1 24.8461,E2 -433.8547} C_DIS
LIN {X -38.2133,Y 9.525,Z 63,A 159.9514,B 24.8413,C -2.9057,E1 24.844,E2 -436.7816} C_DIS
LIN {X -38.695,Y 7.3299,Z 63,A 163.7835,B 24.8418,C -2.9014,E1 24.8419,E2 -440.6259} C_DIS
LIN {X -39.2623,Y 3.0805,Z 63,A 169.8163,B 24.8442,C -2.8797,E1 24.8401,E2 -446.643} C_DIS
LIN {X -39.3826,Y 0.1544,Z 63,A 173.8455,B 24.8459,C -2.864,E1 24.8398,E2 -450.6589} C_DIS
LIN {X -39.335,Y -1.9544,Z 63,A 176.7334,B 24.8471,C -2.8525,E1 24.8401,E2 -453.5367} C_DIS
LIN {X -39.2194,Y -3.5861,Z 63,A 179.059,B 24.848,C -2.8446,E1 24.8406,E2 -455.8573} C_DIS
LIN {X -39.0059,Y -5.4375,Z 63,A -178.0361,B 24.8487,C -2.8383,E1 24.8416,E2 -458.7644} C_DIS
LIN {X -38.6496,Y -7.5656,Z 63,A -174.8921,B 24.8497,C -2.8288,E1 24.8432,E2 -461.9043} C_DIS
LIN {X -38.2184,Y -9.5082,Z 63,A -171.9383,B 24.8505,C -2.8207,E1 24.8451,E2 -464.8561} C_DIS
LIN {X -37.7271,Y -11.3,Z 63,A -169.2856,B 24.8514,C -2.8122,E1 24.8471,E2 -467.5038} C_DIS
LIN {X -37.1287,Y -13.1333,Z 63,A -166.2663,B 24.8521,C -2.8063,E1 24.8499,E2 -470.5262} C_DIS
LIN {X -36.0188,Y -15.9258,Z 63,A -162.1297,B 24.8536,C -2.7916,E1 24.8543,E2 -474.6505} C_DIS
LIN {X -35.07,Y -17.9196,Z 63,A -158.2742,B 24.8538,C -2.7898,E1 24.8591,E2 -478.5225} C_DIS
LIN {X -33.234,Y -21.1316,Z 63,A -152.988,B 24.8554,C -2.7748,E1 24.8667,E2 -483.8003} C_DIS
LIN {X -31.605,Y -23.4973,Z 63,A -149.5915,B 24.8573,C -2.7561,E1 24.8721,E2 -487.1686} C_DIS
LIN {X -30.6024,Y -24.7893,Z 63,A -146.7743,B 24.8573,C -2.7554,E1 24.877,E2 -489.9974} C_DIS
LIN {X -29.4696,Y -26.1265,Z 63,A -144.4151,B 24.8582,C -2.7476,E1 24.8813,E2 -492.3487} C_DIS
LIN {X -27.9547,Y -27.7409,Z 63,A -140.4993,B 24.8581,C -2.7488,E1 24.889,E2 -496.2841} C_DIS
LIN {X -25.8605,Y -29.7028,Z 63,A -136.5984,B 24.8592,C -2.7375,E1 24.897,E2 -500.1737} C_DIS
LIN {X -23.6051,Y -31.5249,Z 63,A -132.1002,B 24.8597,C -2.7335,E1 24.907,E2 -504.6787} C_DIS
LIN {X -20.7367,Y -33.4818,Z 63,A -126.8941,B 24.8603,C -2.7276,E1 24.9191,E2 -509.8878} C_DIS
LIN {X -17.628,Y -35.2177,Z 63,A -122.3637,B 24.8618,C -2.713,E1 24.9302,E2 -514.3961} C_DIS
LIN {X -15.6603,Y -36.1356,Z 63,A -118.709,B 24.8615,C -2.7158,E1 24.9396,E2 -518.0663} C_DIS
LIN {X -12.7756,Y -37.2534,Z 63,A -114.4068,B 24.8621,C -2.7094,E1 24.9509,E2 -522.3619} C_DIS
LIN {X -10.9683,Y -37.8255,Z 63,A -112.089,B 24.8629,C -2.7019,E1 24.957,E2 -524.6657} C_DIS
LIN {X -9.0963,Y -38.3187,Z 63,A -108.8039,B 24.8624,C -2.7064,E1 24.966,E2 -527.9662} C_DIS
LIN {X -7.0819,Y -38.7412,Z 63,A -106.1915,B 24.8631,C -2.7003,E1 24.9731,E2 -530.5669} C_DIS
LIN {X -5.6238,Y -38.9794,Z 63,A -104.1263,B 24.8632,C -2.6986,E1 24.9788,E2 -532.63} C_DIS
LIN {X -3.4345,Y -39.2333,Z 63,A -100.5416,B 24.8628,C -2.7034,E1 24.9888,E2 -536.2281} C_DIS
LIN {X -1.713,Y -39.3457,Z 63,A -97.9709,B 24.8626,C -2.7044,E1 24.996,E2 -538.8019} C_DIS
LIN {X 0.2105,Y -39.3778,Z 63,A -96.0691,B 24.8638,C -2.6928,E1 25.0012,E2 -540.676} C_DIS
Enddeposition()
LIN {X 0.2105,Y -39.3778,Z 63,A -96.0691,B 24.8638,C -2.6928,E1 25.0012,E2 -540.676} C_DIS
Startdeposition()
$VEL.CP = VEL_PRINT
LIN {X -0.7749,Y -38.4251,Z 63,A -98.2522,B 24.8632,C -2.6994,E1 24.9951,E2 -538.5087} C_DIS
LIN {X -2.739,Y -38.3357,Z 63,A -101.1539,B 24.8632,C -2.6997,E1 24.987,E2 -535.6067} C_DIS
LIN {X -4.6334,Y -38.1531,Z 63,A -104.0974,B 24.8632,C -2.6986,E1 24.9789,E2 -532.6589} C_DIS
LIN {X -6.1937,Y -37.9306,Z 63,A -106.4022,B 24.8632,C -2.6998,E1 24.9725,E2 -530.3548} C_DIS
LIN {X -8.0177,Y -37.5879,Z 63,A -109.0555,B 24.8629,C -2.7023,E1 24.9652,E2 -527.7044} C_DIS
LIN {X -9.6045,Y -37.2137,Z 63,A -111.5633,B 24.8629,C -2.7026,E1 24.9584,E2 -525.194} C_DIS
LIN {X -11.3391,Y -36.7224,Z 63,A -114.339,B 24.8628,C -2.7034,E1 24.951,E2 -522.4154} C_DIS
LIN {X -13.4142,Y -36.0164,Z 63,A -117.3271,B 24.8621,C -2.7094,E1 24.9432,E2 -519.4359} C_DIS
LIN {X -15.6083,Y -35.1214,Z 63,A -121.4443,B 24.8625,C -2.7061,E1 24.9325,E2 -515.3013} C_DIS
LIN {X -17.6264,Y -34.1529,Z 63,A -124.2377,B 24.8614,C -2.7164,E1 24.9256,E2 -512.5251} C_DIS
LIN {X -19.0657,Y -33.3708,Z 63,A -127.1521,B 24.8616,C -2.7142,E1 24.9184,E2 -509.597} C_DIS
LIN {X -21.5361,Y -31.8324,Z 63,A -131.797,B 24.8613,C -2.7174,E1 24.9076,E2 -504.9447} C_DIS
LIN {X -24.4276,Y -29.672,Z 63,A -137.3069,B 24.8605,C -2.7255,E1 24.8954,E2 -499.4337} C_DIS
LIN {X -26.1557,Y -28.1599,Z 63,A -140.556,B 24.8596,C -2.734,E1 24.8888,E2 -496.1919} C_DIS
LIN {X -28.3313,Y -25.97,Z 63,A -144.7267,B 24.8581,C -2.7483,E1 24.8807,E2 -492.0372} C_DIS
LIN {X -30.1751,Y -23.8027,Z 63,A -148.9586,B 24.8571,C -2.758,E1 24.8732,E2 -487.809} C_DIS
LIN {X -31.5723,Y -21.9157,Z 63,A -153.0925,B 24.8569,C -2.76,E1 24.8665,E2 -483.6596} C_DIS
LIN {X -33.4083,Y -19.0004,Z 63,A -157.9698,B 24.8553,C -2.7758,E1 24.8595,E2 -478.7951} C_DIS
LIN {X -34.4446,Y -17.0491,Z 63,A -161.4223,B 24.8545,C -2.7831,E1 24.8551,E2 -475.3415} C_DIS
LIN {X -35.8694,Y -13.8034,Z 63,A -166.218,B 24.8524,C -2.8027,E1 24.8499,E2 -470.5662} C_DIS
LIN {X -36.4973,Y -12.0447,Z 63,A -169.1097,B 24.8517,C -2.8097,E1 24.8473,E2 -467.6747} C_DIS
LIN {X -36.9807,Y -10.4656,Z 63,A -171.3725,B 24.8507,C -2.8189,E1 24.8455,E2 -465.4209} C_DIS
LIN {X -37.3489,Y -9.0646,Z 63,A -173.5162,B 24.85,C -2.8255,E1 24.844,E2 -463.2804} C_DIS
LIN {X -37.7528,Y -7.1993,Z 63,A -177.0624,B 24.8498,C -2.8273,E1 24.8421,E2 -459.7177} C_DIS
LIN {X -38.2256,Y -3.9883,Z 63,A 178.2448,B 24.8481,C -2.8436,E1 24.8404,E2 -455.0358} C_DIS
LIN {X -38.3814,Y -1.9975,Z 63,A 175.6417,B 24.8467,C -2.8564,E1 24.8399,E2 -452.4477} C_DIS
LIN {X -38.4309,Y -0.4633,Z 63,A 173.2899,B 24.846,C -2.8629,E1 24.8398,E2 -450.0974} C_DIS
LIN {X -38.4131,Y 1.2434,Z 63,A 170.583,B 24.8453,C -2.8694,E1 24.8399,E2 -447.3895} C_DIS
LIN {X -38.317,Y 2.9859,Z 63,A 167.8864,B 24.8445,C -2.8766,E1 24.8405,E2 -444.6941} C_DIS
LIN {X -38.0154,Y 5.6543,Z 63,A 163.5685,B 24.8435,C -2.8862,E1 24.842,E2 -440.3732} C_DIS
LIN {X -37.613,Y 7.8992,Z 63,A 160.627,B 24.8419,C -2.9011,E1 24.8436,E2 -437.4501} C_DIS
LIN {X -37.1358,Y 9.9021,Z 63,A 157.2365,B 24.8412,C -2.9075,E1 24.8459,E2 -434.0551} C_DIS
LIN {X -36.413,Y 12.2959,Z 63,A 153.6011,B 24.8398,C -2.9197,E1 24.849,E2 -430.4281} C_DIS
LIN {X -35.4597,Y 14.8233,Z 63,A 150.1834,B 24.8378,C -2.9377,E1 24.8524,E2 -427.0342} C_DIS
LIN {X -34.5727,Y 16.7887,Z 63,A 145.7517,B 24.8381,C -2.9352,E1 24.8577,E2 -422.5725} C_DIS
LIN {X -33.4388,Y 18.9474,Z 63,A 142.0945,B 24.837,C -2.9453,E1 24.8626,E2 -418.9202} C_DIS
LIN {X -31.4988,Y 22.0206,Z 63,A 137.3766,B 24.8346,C -2.967,E1 24.8698,E2 -414.2305} C_DIS
LIN {X -30.6641,Y 23.1696,Z 63,A 135.1001,B 24.8341,C -2.9709,E1 24.8736,E2 -411.9524} C_DIS
LIN {X -29.1028,Y 25.1035,Z 63,A 131.0224,B 24.8335,C -2.9765,E1 24.8809,E2 -407.8694} C_DIS
LIN {X -27.3951,Y 26.9559,Z 63,A 127.5921,B 24.8321,C -2.9889,E1 24.8875,E2 -404.4537} C_DIS
LIN {X -25.5936,Y 28.6719,Z 63,A 123.6009,B 24.8315,C -2.9944,E1 24.8957,E2 -400.4595} C_DIS
LIN {X -23.7016,Y 30.255,Z 63,A 120.2842,B 24.8302,C -3.0059,E1 24.9028,E2 -397.158} C_DIS
LIN {X -22.3422,Y 31.2719,Z 63,A 117.247,B 24.8302,C -3.0056,E1 24.9097,E2 -394.1094} C_DIS
LIN {X -19.5587,Y 33.0842,Z 63,A 112.9991,B 24.8283,C -3.0223,E1 24.9197,E2 -389.8878} C_DIS
LIN {X -18.3526,Y 33.7682,Z 63,A 110.8504,B 24.828,C -3.0249,E1 24.9249,E2 -387.7391} C_DIS
LIN {X -16.8689,Y 34.5331,Z 63,A 107.75,B 24.8283,C -3.022,E1 24.9327,E2 -384.6237} C_DIS
LIN {X -14.8085,Y 35.4659,Z 63,A 104.6863,B 24.8274,C -3.0303,E1 24.9405,E2 -381.5724} C_DIS
LIN {X -12.6532,Y 36.2906,Z 63,A 101.177,B 24.827,C -3.0338,E1 24.9497,E2 -378.0644} C_DIS
LIN {X -10.5867,Y 36.9464,Z 63,A 98.0027,B 24.8265,C -3.038,E1 24.9582,E2 -374.8948} C_DIS
LIN {X -8.5329,Y 37.474,Z 63,A 94.8908,B 24.8261,C -3.0415,E1 24.9666,E2 -371.7869} C_DIS
LIN {X -5.7032,Y 38.0071,Z 63,A 89.6231,B 24.8271,C -3.033,E1 24.9812,E2 -366.494} C_DIS
LIN {X -1.828,Y 38.3899,Z 63,A 84.4607,B 24.8259,C -3.0433,E1 24.9955,E2 -361.3539} C_DIS
LIN {X 0.7724,Y 38.4254,Z 63,A 80.9414,B 24.8253,C -3.0485,E1 25.0053,E2 -357.8471} C_DIS
LIN {X 2.5628,Y 38.3476,Z 63,A 78.4707,B 24.825,C -3.0511,E1 25.0122,E2 -355.3835} C_DIS
LIN {X 3.9489,Y 38.2297,Z 63,A 76.0267,B 24.8256,C -3.0461,E1 25.019,E2 -352.9292} C_DIS
LIN {X 6.2989,Y 37.9134,Z 63,A 72.5617,B 24.8256,C -3.0461,E1 25.0286,E2 -349.4673} C_DIS
LIN {X 8.2972,Y 37.527,Z 63,A 69.5665,B 24.8256,C -3.0452,E1 25.0367,E2 -346.4738} C_DIS
LIN {X 10.3975,Y 36.9999,Z 63,A 66.6205,B 24.8255,C -3.047,E1 25.0447,E2 -343.5367} C_DIS
LIN {X 12.3909,Y 36.3808,Z 63,A 62.9968,B 24.8265,C -3.0377,E1 25.0543,E2 -339.8976} C_DIS
LIN {X 14.1401,Y 35.7375,Z 63,A 60.1634,B 24.8269,C -3.0343,E1 25.0617,E2 -337.0624} C_DIS
LIN {X 16.6598,Y 34.6342,Z 63,A 56.3199,B 24.8271,C -3.0333,E1 25.0715,E2 -333.2261} C_DIS
LIN {X 17.9721,Y 33.9722,Z 63,A 53.9457,B 24.8277,C -3.0279,E1 25.0774,E2 -330.8458} C_DIS
LIN {X 20.5513,Y 32.4777,Z 63,A 49.8011,B 24.8279,C -3.0257,E1 25.0873,E2 -326.7088} C_DIS
LIN {X 22.0941,Y 31.4482,Z 63,A 47.0656,B 24.8284,C -3.0217,E1 25.0936,E2 -323.9731} C_DIS
LIN {X 23.669,Y 30.2807,Z 63,A 44.5036,B 24.8284,C -3.0219,E1 25.0993,E2 -321.4208} C_DIS
LIN {X 24.8528,Y 29.3164,Z 63,A 41.7911,B 24.8296,C -3.0113,E1 25.1051,E2 -318.6937} C_DIS
LIN {X 26.3517,Y 27.9766,Z 63,A 38.9285,B 24.83,C -3.0074,E1 25.111,E2 -315.8333} C_DIS
LIN {X 27.5558,Y 26.7912,Z 63,A 36.4224,B 24.8306,C -3.0024,E1 25.1159,E2 -313.3259} C_DIS
LIN {X 28.82,Y 25.4273,Z 63,A 33.7228,B 24.8311,C -2.9974,E1 25.121,E2 -310.6265} C_DIS
LIN {X 29.8282,Y 24.236,Z 63,A 30.9484,B 24.8325,C -2.9853,E1 25.126,E2 -307.8364} C_DIS
LIN {X 31.0636,Y 22.6311,Z 63,A 27.9563,B 24.8333,C -2.9785,E1 25.1309,E2 -304.8424} C_DIS
LIN {X 32.583,Y 20.3824,Z 63,A 24.3281,B 24.8337,C -2.9748,E1 25.1365,E2 -301.2233} C_DIS
LIN {X 33.3085,Y 19.1741,Z 63,A 22.1264,B 24.8345,C -2.9677,E1 25.1396,E2 -299.0164} C_DIS
LIN {X 34.2465,Y 17.4438,Z 63,A 19.5555,B 24.8347,C -2.9655,E1 25.1429,E2 -296.4538} C_DIS
LIN {X 34.7791,Y 16.3563,Z 63,A 17.2797,B 24.8361,C -2.9533,E1 25.1457,E2 -294.1612} C_DIS
LIN {X 35.7658,Y 14.0681,Z 63,A 13.5006,B 24.8374,C -2.9418,E1 25.1497,E2 -290.3758} C_DIS
LIN {X 36.4894,Y 12.0696,Z 63,A 10.4973,B 24.8381,C -2.9352,E1 25.1524,E2 -287.3738} C_DIS
LIN {X 37.1348,Y 9.9058,Z 63,A 7.2612,B 24.839,C -2.9273,E1 25.1549,E2 -284.1375} C_DIS
LIN {X 37.684,Y 7.5533,Z 63,A 3.4162,B 24.8406,C -2.9126,E1 25.1572,E2 -280.2801} C_DIS
LIN {X 38.0425,Y 5.4661,Z 63,A -0.0187,B 24.8421,C -2.8985,E1 25.1586,E2 -276.832} C_DIS
LIN {X 38.397,Y 1.6657,Z 63,A -4.8675,B 24.8426,C -2.8942,E1 25.1597,E2 -272.002} C_DIS
LIN {X 38.4328,Y 0.0494,Z 63,A -7.7741,B 24.8443,C -2.8788,E1 25.1597,E2 -269.076} C_DIS
LIN {X 38.3433,Y -2.6255,Z 63,A -11.3836,B 24.845,C -2.8723,E1 25.1593,E2 -265.4726} C_DIS
LIN {X 38.1814,Y -4.3915,Z 63,A -14.2731,B 24.8463,C -2.8601,E1 25.1584,E2 -262.5714} C_DIS
LIN {X 37.83,Y -6.7821,Z 63,A -18.2153,B 24.8481,C -2.8434,E1 25.1566,E2 -258.6128} C_DIS
LIN {X 36.9383,Y -10.6153,Z 63,A -23.5665,B 24.8492,C -2.8335,E1 25.153,E2 -253.269} C_DIS
LIN {X 36.2185,Y -12.8588,Z 63,A -27.1933,B 24.8505,C -2.821,E1 25.1497,E2 -249.6331} C_DIS
LIN {X 35.4255,Y -14.9043,Z 63,A -30.0461,B 24.8508,C -2.8179,E1 25.1468,E2 -246.7887} C_DIS
LIN {X 34.6251,Y -16.6795,Z 63,A -33.1429,B 24.8521,C -2.8063,E1 25.1431,E2 -243.6811} C_DIS
LIN {X 33.6049,Y -18.6494,Z 63,A -36.6679,B 24.8534,C -2.7934,E1 25.1384,E2 -240.1441} C_DIS
LIN {X 32.5937,Y -20.3655,Z 63,A -39.8105,B 24.8546,C -2.7824,E1 25.1338,E2 -236.9915} C_DIS
LIN {X 30.9353,Y -22.8063,Z 63,A -43.6582,B 24.8549,C -2.7791,E1 25.1276,E2 -233.1549} C_DIS
LIN {X 29.7882,Y -24.2854,Z 63,A -46.2364,B 24.8553,C -2.7752,E1 25.1232,E2 -230.5794} C_DIS
LIN {X 28.9545,Y -25.2733,Z 63,A -48.5398,B 24.8565,C -2.7645,E1 25.119,E2 -228.2612} C_DIS
LIN {X 27.3091,Y -27.0421,Z 63,A -51.6462,B 24.8565,C -2.7634,E1 25.113,E2 -225.1656} C_DIS
LIN {X 26.3555,Y -27.973,Z 63,A -53.7068,B 24.8572,C -2.7576,E1 25.1088,E2 -223.0999} C_DIS
LIN {X 25.418,Y -28.8266,Z 63,A -55.9653,B 24.8582,C -2.7478,E1 25.1041,E2 -220.827} C_DIS
LIN {X 23.5829,Y -30.3474,Z 63,A -59.1576,B 24.8584,C -2.7455,E1 25.0972,E2 -217.6415} C_DIS
LIN {X 22.5134,Y -31.1495,Z 63,A -61.3324,B 24.8591,C -2.7388,E1 25.0923,E2 -215.4584} C_DIS
LIN {X 21.0542,Y -32.1534,Z 63,A -64.2121,B 24.86,C -2.7301,E1 25.0856,E2 -212.5678} C_DIS
LIN {X 18.7467,Y -33.5509,Z 63,A -67.7021,B 24.86,C -2.7307,E1 25.0772,E2 -209.09} C_DIS
LIN {X 16.945,Y -34.4961,Z 63,A -70.8031,B 24.8606,C -2.7248,E1 25.0695,E2 -205.9834} C_DIS
LIN {X 15.7455,Y -35.0598,Z 63,A -73.1714,B 24.8614,C -2.7162,E1 25.0634,E2 -203.6006} C_DIS
LIN {X 13.4273,Y -36.0118,Z 63,A -76.8004,B 24.8618,C -2.7126,E1 25.054,E2 -199.9712} C_DIS
LIN {X 11.6289,Y -36.632,Z 63,A -79.4194,B 24.8618,C -2.7122,E1 25.0471,E2 -197.3564} C_DIS
LIN {X 9.9215,Y -37.1306,Z 63,A -82.2297,B 24.8624,C -2.7072,E1 25.0395,E2 -194.5388} C_DIS
LIN {X 8.0286,Y -37.5852,Z 63,A -85.6403,B 24.8633,C -2.6976,E1 25.0301,E2 -191.1099} C_DIS
LIN {X 4.8271,Y -38.1289,Z 63,A -90.2923,B 24.8634,C -2.6969,E1 25.0173,E2 -186.4604} C_DIS
LIN {X 1.6498,Y -38.3974,Z 63,A -94.6658,B 24.8631,C -2.6998,E1 25.0052,E2 -182.0959} C_DIS
LIN {X 0.2034,Y -38.431,Z 63,A -95.9932,B 24.8621,C -2.7102,E1 25.0015,E2 -180.7934} C_DIS
Enddeposition()
LIN {X 0.2034,Y -38.431,Z 63,A -95.9932,B 24.8621,C -2.7102,E1 25.0015,E2 -180.7934} C_DIS
Startdeposition()
$VEL.CP = VEL_PRINT
LIN {X 0.6697,Y -37.4773,Z 63,A -93.7957,B 24.8583,C -2.7464,E1 25.0079,E2 -183.0764} C_DIS
LIN {X 4.651,Y -37.194,Z 63,A -88.4347,B 24.859,C -2.7395,E1 25.0227,E2 -188.418} C_DIS
LIN {X 7.1919,Y -36.7864,Z 63,A -84.8526,B 24.8592,C -2.7378,E1 25.0326,E2 -191.9921} C_DIS
LIN {X 8.7011,Y -36.4599,Z 63,A -81.6992,B 24.8579,C -2.751,E1 25.0412,E2 -195.1723} C_DIS
LIN {X 12.4252,Y -35.364,Z 63,A -76.4634,B 24.8582,C -2.748,E1 25.0551,E2 -200.3915} C_DIS
LIN {X 14.6038,Y -34.5214,Z 63,A -72.6414,B 24.8573,C -2.7565,E1 25.065,E2 -204.225} C_DIS
LIN {X 16.6312,Y -33.5917,Z 63,A -69.4175,B 24.857,C -2.7591,E1 25.0731,E2 -207.4467} C_DIS
LIN {X 18.2654,Y -32.7318,Z 63,A -66.7771,B 24.8568,C -2.7612,E1 25.0796,E2 -210.0846} C_DIS
LIN {X 19.851,Y -31.7952,Z 63,A -63.7909,B 24.856,C -2.7689,E1 25.0868,E2 -213.0797} C_DIS
LIN {X 21.2916,Y -30.8493,Z 63,A -61.4244,B 24.8559,C -2.77,E1 25.0922,E2 -215.4408} C_DIS
LIN {X 22.5972,Y -29.906,Z 63,A -58.8641,B 24.8552,C -2.7765,E1 25.098,E2 -218.0075} C_DIS
LIN {X 24.3808,Y -28.4707,Z 63,A -54.7239,B 24.8534,C -2.7938,E1 25.1069,E2 -222.1728} C_DIS
LIN {X 26.9642,Y -26.0371,Z 63,A -49.4899,B 24.8523,C -2.8037,E1 25.1173,E2 -227.4081} C_DIS
LIN {X 28.5312,Y -24.3098,Z 63,A -46.3891,B 24.8522,C -2.8054,E1 25.123,E2 -230.4991} C_DIS
LIN {X 29.5724,Y -23.0327,Z 63,A -43.9944,B 24.8517,C -2.8101,E1 25.1272,E2 -232.8936} C_DIS
LIN {X 30.6787,Y -21.5371,Z 63,A -40.8359,B 24.8503,C -2.8226,E1 25.1324,E2 -236.0663} C_DIS
LIN {X 31.6781,Y -20.0385,Z 63,A -38.4821,B 24.8502,C -2.8239,E1 25.1359,E2 -238.4114} C_DIS
LIN {X 32.6014,Y -18.4978,Z 63,A -35.167,B 24.8484,C -2.8406,E1 25.1406,E2 -241.7491} C_DIS
LIN {X 33.9184,Y -15.955,Z 63,A -31.0407,B 24.8475,C -2.8493,E1 25.1457,E2 -245.8739} C_DIS
LIN {X 34.6777,Y -14.229,Z 63,A -28.1636,B 24.8466,C -2.8578,E1 25.1488,E2 -248.7554} C_DIS
LIN {X 35.55,Y -11.883,Z 63,A -24.2559,B 24.8452,C -2.8707,E1 25.1525,E2 -252.6716} C_DIS
LIN {X 36.225,Y -9.6286,Z 63,A -20.4671,B 24.8436,C -2.8848,E1 25.1553,E2 -256.4722} C_DIS
LIN {X 36.9003,Y -6.5852,Z 63,A -15.8558,B 24.8423,C -2.8972,E1 25.1578,E2 -261.0857} C_DIS
LIN {X 37.3247,Y -3.4414,Z 63,A -11.4004,B 24.8413,C -2.9061,E1 25.1593,E2 -265.5359} C_DIS
LIN {X 37.4472,Y -1.644,Z 63,A -8.8154,B 24.8407,C -2.912,E1 25.1597,E2 -268.1196} C_DIS
LIN {X 37.4742,Y 0.8398,Z 63,A -4.7664,B 24.8389,C -2.9279,E1 25.1597,E2 -272.1821} C_DIS
LIN {X 37.2901,Y 3.8021,Z 63,A -0.0618,B 24.837,C -2.9447,E1 25.1586,E2 -276.8985} C_DIS
LIN {X 37.0183,Y 5.8882,Z 63,A 2.6379,B 24.8369,C -2.9464,E1 25.1575,E2 -279.5863} C_DIS
LIN {X 36.5896,Y 8.1378,Z 63,A 5.8898,B 24.8361,C -2.953,E1 25.1558,E2 -282.835} C_DIS
LIN {X 36.1994,Y 9.7262,Z 63,A 8.8961,B 24.8344,C -2.9685,E1 25.1536,E2 -285.8606} C_DIS
LIN {X 35.4857,Y 12.0737,Z 63,A 12.7641,B 24.833,C -2.9813,E1 25.1503,E2 -289.7368} C_DIS
LIN {X 34.6924,Y 14.1929,Z 63,A 15.8943,B 24.8324,C -2.9859,E1 25.1471,E2 -292.8608} C_DIS
LIN {X 34.0607,Y 15.6493,Z 63,A 18.1192,B 24.832,C -2.9895,E1 25.1446,E2 -295.0821} C_DIS
LIN {X 33.3335,Y 17.1429,Z 63,A 20.8348,B 24.8309,C -2.9991,E1 25.1412,E2 -297.8059} C_DIS
LIN {X 32.1736,Y 19.2325,Z 63,A 24.9548,B 24.829,C -3.0159,E1 25.1354,E2 -301.9443} C_DIS
LIN {X 30.3361,Y 22.0168,Z 63,A 29.7321,B 24.8282,C -3.0235,E1 25.1279,E2 -306.7162} C_DIS
LIN {X 28.3175,Y 24.5587,Z 63,A 34.8776,B 24.8266,C -3.0376,E1 25.1187,E2 -311.8714} C_DIS
LIN {X 26.5612,Y 26.4476,Z 63,A 38.0666,B 24.8269,C -3.0348,E1 25.1126,E2 -315.04} C_DIS
LIN {X 25.6751,Y 27.3091,Z 63,A 40.0563,B 24.8263,C -3.0401,E1 25.1086,E2 -317.0339} C_DIS
LIN {X 24.1659,Y 28.6538,Z 63,A 43.6776,B 24.8247,C -3.0537,E1 25.1009,E2 -320.6734} C_DIS
LIN {X 21.8491,Y 30.4569,Z 63,A 47.9628,B 24.8242,C -3.0585,E1 25.0913,E2 -324.9545} C_DIS
LIN {X 20.0725,Y 31.6565,Z 63,A 50.7724,B 24.8243,C -3.0569,E1 25.0848,E2 -327.7511} C_DIS
LIN {X 18.23,Y 32.7516,Z 63,A 54.5265,B 24.823,C -3.0682,E1 25.0757,E2 -331.5207} C_DIS
LIN {X 15.5179,Y 34.1199,Z 63,A 59.8776,B 24.8212,C -3.0835,E1 25.0622,E2 -336.8943} C_DIS
LIN {X 11.9427,Y 35.5298,Z 63,A 65.0246,B 24.8218,C -3.0788,E1 25.0487,E2 -342.0192} C_DIS
LIN {X 9.6135,Y 36.2294,Z 63,A 68.4566,B 24.8219,C -3.0775,E1 25.0395,E2 -345.4424} C_DIS
LIN {X 8.0982,Y 36.5982,Z 63,A 71.18,B 24.8213,C -3.0832,E1 25.0321,E2 -348.1755} C_DIS
LIN {X 5.2943,Y 37.1075,Z 63,A 75.7944,B 24.8207,C -3.0879,E1 25.0194,E2 -352.7966} C_DIS
LIN {X 2.4006,Y 37.4065,Z 63,A 79.5702,B 24.8217,C -3.0797,E1 25.0089,E2 -356.5507} C_DIS
LIN {X 0.9507,Y 37.4717,Z 63,A 81.8704,B 24.8216,C -3.0805,E1 25.0025,E2 -358.8522} C_DIS
LIN {X -0.5764,Y 37.479,Z 63,A 84.2879,B 24.8216,C -3.0811,E1 24.9957,E2 -361.2711} C_DIS
LIN {X -2.5242,Y 37.3982,Z 63,A 87.0857,B 24.8219,C -3.0778,E1 24.988,E2 -364.0618} C_DIS
LIN {X -4.4772,Y 37.2151,Z 63,A 90.6683,B 24.8213,C -3.0832,E1 24.978,E2 -367.6597} C_DIS
LIN {X -7.3789,Y 36.7502,Z 63,A 94.6288,B 24.8224,C -3.0736,E1 24.9671,E2 -371.6012} C_DIS
LIN {X -8.7813,Y 36.4399,Z 63,A 97.2199,B 24.8221,C -3.0763,E1 24.9601,E2 -374.2021} C_DIS
LIN {X -11.3726,Y 35.7168,Z 63,A 100.6631,B 24.8235,C -3.0642,E1 24.9509,E2 -377.6221} C_DIS
LIN {X -12.9976,Y 35.1579,Z 63,A 103.8404,B 24.8231,C -3.0672,E1 24.9425,E2 -380.8128} C_DIS
LIN {X -14.5578,Y 34.5408,Z 63,A 106.5099,B 24.8234,C -3.0649,E1 24.9356,E2 -383.4828} C_DIS
LIN {X -17.2643,Y 33.2713,Z 63,A 111.4733,B 24.8237,C -3.0621,E1 24.9232,E2 -388.4527} C_DIS
LIN {X -19.8294,Y 31.8087,Z 63,A 115.3819,B 24.8254,C -3.0476,E1 24.9138,E2 -392.3384} C_DIS
LIN {X -21.5113,Y 30.6966,Z 63,A 118.8249,B 24.8256,C -3.0455,E1 24.9059,E2 -395.7881} C_DIS
LIN {X -23.042,Y 29.5653,Z 63,A 121.3718,B 24.8268,C -3.0357,E1 24.9003,E2 -398.3207} C_DIS
LIN {X -24.8785,Y 28.0371,Z 63,A 125.6021,B 24.827,C -3.0338,E1 24.8913,E2 -402.5629} C_DIS
LIN {X -26.7383,Y 26.2692,Z 63,A 129.0655,B 24.8286,C -3.0199,E1 24.8844,E2 -406.0077} C_DIS
LIN {X -28.5414,Y 24.2979,Z 63,A 133.8158,B 24.829,C -3.0166,E1 24.8756,E2 -410.7713} C_DIS
LIN {X -29.9846,Y 22.4927,Z 63,A 136.8296,B 24.8306,C -3.0022,E1 24.8706,E2 -413.765} C_DIS
LIN {X -30.9299,Y 21.1736,Z 63,A 139.5646,B 24.8311,C -2.998,E1 24.8662,E2 -416.5036} C_DIS
LIN {X -32.4997,Y 18.6752,Z 63,A 143.4866,B 24.8331,C -2.9797,E1 24.8605,E2 -420.4019} C_DIS
LIN {X -33.5942,Y 16.626,Z 63,A 148.0549,B 24.8331,C -2.9795,E1 24.8547,E2 -424.994} C_DIS
LIN {X -34.6398,Y 14.3221,Z 63,A 151.9256,B 24.8344,C -2.9681,E1 24.8505,E2 -428.8589} C_DIS
LIN {X -35.8126,Y 11.0658,Z 63,A 156.6199,B 24.8369,C -2.9463,E1 24.8463,E2 -433.5278} C_DIS
LIN {X -36.3981,Y 8.9544,Z 63,A 160.0937,B 24.8379,C -2.9372,E1 24.8439,E2 -437} C_DIS
LIN {X -36.8362,Y 6.9362,Z 63,A 163.1268,B 24.8391,C -2.9262,E1 24.8422,E2 -440.0247} C_DIS
LIN {X -37.1233,Y 5.1795,Z 63,A 166.0254,B 24.8398,C -2.9194,E1 24.841,E2 -442.9243} C_DIS
LIN {X -37.3799,Y 2.789,Z 63,A 169.4292,B 24.8414,C -2.9053,E1 24.8401,E2 -446.3148} C_DIS
LIN {X -37.4618,Y 1.2746,Z 63,A 171.7985,B 24.8421,C -2.8985,E1 24.8398,E2 -448.6822} C_DIS
LIN {X -37.48,Y -0.5221,Z 63,A 174.6602,B 24.843,C -2.891,E1 24.8398,E2 -451.5431} C_DIS
LIN {X -37.3969,Y -2.5433,Z 63,A 177.8759,B 24.8439,C -2.8826,E1 24.8403,E2 -454.758} C_DIS
LIN {X -37.1735,Y -4.8092,Z 63,A -178.9651,B 24.8454,C -2.8688,E1 24.8413,E2 -457.9029} C_DIS
LIN {X -36.8917,Y -6.6329,Z 63,A -175.9954,B 24.8462,C -2.8616,E1 24.8426,E2 -460.873} C_DIS
LIN {X -36.5711,Y -8.2217,Z 63,A -173.4489,B 24.8469,C -2.8548,E1 24.8441,E2 -463.4183} C_DIS
LIN {X -35.8517,Y -10.9399,Z 63,A -168.2906,B 24.8473,C -2.8505,E1 24.8481,E2 -468.5962} C_DIS
LIN {X -35.1392,Y -13.0492,Z 63,A -165.4264,B 24.849,C -2.8354,E1 24.8508,E2 -471.4404} C_DIS
LIN {X -34.1653,Y -15.4184,Z 63,A -161.6317,B 24.8503,C -2.8233,E1 24.855,E2 -475.2271} C_DIS
LIN {X -33.4357,Y -16.943,Z 63,A -159.2791,B 24.8512,C -2.814,E1 24.8578,E2 -477.5702} C_DIS
LIN {X -32.631,Y -18.4444,Z 63,A -156.2019,B 24.8515,C -2.8119,E1 24.862,E2 -480.6586} C_DIS
LIN {X -31.7621,Y -19.904,Z 63,A -153.4724,B 24.852,C -2.8066,E1 24.866,E2 -483.3895} C_DIS
LIN {X -30.2683,Y -22.1092,Z 63,A -150.2293,B 24.854,C -2.7882,E1 24.8712,E2 -486.6044} C_DIS
LIN {X -29.2586,Y -23.4303,Z 63,A -147.1787,B 24.854,C -2.7875,E1 24.8764,E2 -489.6678} C_DIS
LIN {X -28.0081,Y -24.911,Z 63,A -144.514,B 24.8551,C -2.7778,E1 24.8813,E2 -492.3215} C_DIS
LIN {X -27.0254,Y -25.9736,Z 63,A -142.1033,B 24.8553,C -2.7752,E1 24.8859,E2 -494.7364} C_DIS
LIN {X -25.8506,Y -27.1435,Z 63,A -139.4707,B 24.8558,C -2.7711,E1 24.8912,E2 -497.3702} C_DIS
LIN {X -24.6293,Y -28.2559,Z 63,A -136.6363,B 24.8559,C -2.7697,E1 24.8971,E2 -500.2124} C_DIS
LIN {X -22.4464,Y -30.0193,Z 63,A -132.9956,B 24.8574,C -2.755,E1 24.905,E2 -503.8315} C_DIS
LIN {X -20.9122,Y -31.1077,Z 63,A -129.608,B 24.8574,C -2.7561,E1 24.9128,E2 -507.2332} C_DIS
LIN {X -19.1601,Y -32.2164,Z 63,A -126.2252,B 24.8576,C -2.7539,E1 24.9209,E2 -510.6214} C_DIS
LIN {X -16.5724,Y -33.6208,Z 63,A -122.3542,B 24.8589,C -2.741,E1 24.9304,E2 -514.4722} C_DIS
LIN {X -14.725,Y -34.47,Z 63,A -118.8561,B 24.8588,C -2.7422,E1 24.9394,E2 -517.9818} C_DIS
LIN {X -12.6641,Y -35.2792,Z 63,A -115.5999,B 24.8592,C -2.7377,E1 24.9479,E2 -521.2339} C_DIS
LIN {X -11.1392,Y -35.7899,Z 63,A -112.9199,B 24.8592,C -2.7385,E1 24.955,E2 -523.9208} C_DIS
LIN {X -8.8103,Y -36.4332,Z 63,A -109.647,B 24.8599,C -2.7313,E1 24.9638,E2 -527.1813} C_DIS
LIN {X -7.4904,Y -36.7271,Z 63,A -107.2145,B 24.8595,C -2.7349,E1 24.9705,E2 -529.6254} C_DIS
LIN {X -5.516,Y -37.0758,Z 63,A -104.2729,B 24.8598,C -2.7325,E1 24.9786,E2 -532.5639} C_DIS
LIN {X -3.7976,Y -37.2906,Z 63,A -101.8319,B 24.8601,C -2.7295,E1 24.9854,E2 -534.9995} C_DIS
LIN {X -2.5791,Y -37.3945,Z 63,A -99.4449,B 24.8594,C -2.7362,E1 24.9921,E2 -537.4033} C_DIS
LIN {X 0.1925,Y -37.4828,Z 63,A -95.8127,B 24.8601,C -2.729,E1 25.0021,E2 -541.0186} C_DIS
Enddeposition()
LIN {X 0.1925,Y -37.4828,Z 63,A -95.8127,B 24.8601,C -2.729,E1 25.0021,E2 -541.0186} C_DIS
Startdeposition()
$VEL.CP = VEL_PRINT
LIN {X -0.3338,Y -36.5321,Z 63,A -97.8473,B 24.8601,C -2.73,E1 24.9965,E2 -538.9864} C_DIS
LIN {X -2.4193,Y -36.4533,Z 63,A -100.8459,B 24.8597,C -2.7331,E1 24.9881,E2 -535.9945} C_DIS
LIN {X -3.9798,Y -36.316,Z 63,A -103.2912,B 24.8597,C -2.7335,E1 24.9813,E2 -533.5486} C_DIS
LIN {X -5.3546,Y -36.1395,Z 63,A -105.9111,B 24.8602,C -2.7286,E1 24.974,E2 -530.915} C_DIS
LIN {X -8.0086,Y -35.6453,Z 63,A -109.7534,B 24.8595,C -2.7349,E1 24.9636,E2 -527.0832} C_DIS
LIN {X -9.8734,Y -35.1741,Z 63,A -113.0259,B 24.8596,C -2.7337,E1 24.9547,E2 -523.803} C_DIS
LIN {X -11.9096,Y -34.5377,Z 63,A -116.8857,B 24.86,C -2.7305,E1 24.9444,E2 -519.9283} C_DIS
LIN {X -14.0248,Y -33.7347,Z 63,A -120.146,B 24.8593,C -2.7371,E1 24.936,E2 -516.6766} C_DIS
LIN {X -16.3883,Y -32.6519,Z 63,A -123.5259,B 24.858,C -2.7494,E1 24.9275,E2 -513.3175} C_DIS
LIN {X -17.6201,Y -32.0038,Z 63,A -125.9949,B 24.858,C -2.7491,E1 24.9215,E2 -510.8407} C_DIS
LIN {X -18.9509,Y -31.2339,Z 63,A -128.2943,B 24.8576,C -2.7536,E1 24.9159,E2 -508.5454} C_DIS
LIN {X -20.2827,Y -30.3861,Z 63,A -131.2647,B 24.8577,C -2.7522,E1 24.909,E2 -505.5618} C_DIS
LIN {X -21.7692,Y -29.3401,Z 63,A -134.0704,B 24.8572,C -2.7574,E1 24.9026,E2 -502.7586} C_DIS
LIN {X -23.5429,Y -27.9355,Z 63,A -137.1489,B 24.856,C -2.7686,E1 24.896,E2 -499.6954} C_DIS
LIN {X -24.4926,Y -27.1078,Z 63,A -139.8726,B 24.8564,C -2.7648,E1 24.8903,E2 -496.9517} C_DIS
LIN {X -26.7912,Y -24.8387,Z 63,A -144.2097,B 24.8546,C -2.7826,E1 24.8819,E2 -492.6386} C_DIS
LIN {X -28.1926,Y -23.235,Z 63,A -148.1766,B 24.8544,C -2.7839,E1 24.8746,E2 -488.6567} C_DIS
LIN {X -29.424,Y -21.6547,Z 63,A -150.7744,B 24.8531,C -2.7966,E1 24.8703,E2 -486.0769} C_DIS
LIN {X -30.3271,Y -20.3709,Z 63,A -153.7593,B 24.853,C -2.7977,E1 24.8656,E2 -483.0796} C_DIS
LIN {X -31.2692,Y -18.8929,Z 63,A -156.3333,B 24.8521,C -2.8063,E1 24.8618,E2 -480.5132} C_DIS
LIN {X -32.2041,Y -17.2515,Z 63,A -159.1768,B 24.8511,C -2.8152,E1 24.858,E2 -477.6761} C_DIS
LIN {X -33.0176,Y -15.6388,Z 63,A -162.4031,B 24.8507,C -2.8193,E1 24.854,E2 -474.442} C_DIS
LIN {X -34.0345,Y -13.2798,Z 63,A -166.2568,B 24.8493,C -2.8322,E1 24.8499,E2 -470.5977} C_DIS
LIN {X -34.7748,Y -11.1985,Z 63,A -169.4153,B 24.8479,C -2.845,E1 24.8471,E2 -467.4519} C_DIS
LIN {X -35.2216,Y -9.7029,Z 63,A -172.1177,B 24.8474,C -2.8499,E1 24.845,E2 -464.7456} C_DIS
LIN {X -35.7222,Y -7.6553,Z 63,A -175.6756,B 24.8466,C -2.8576,E1 24.8428,E2 -461.1852} C_DIS
LIN {X -36.1495,Y -5.2843,Z 63,A -179.0221,B 24.8449,C -2.873,E1 24.8413,E2 -457.8556} C_DIS
LIN {X -36.3172,Y -3.9676,Z 63,A 178.8504,B 24.8443,C -2.879,E1 24.8406,E2 -455.7298} C_DIS
LIN {X -36.4545,Y -2.4015,Z 63,A 176.3445,B 24.8435,C -2.8863,E1 24.84,E2 -453.2263} C_DIS
LIN {X -36.5325,Y 0.2485,Z 63,A 172.3346,B 24.8419,C -2.9006,E1 24.8398,E2 -449.2264} C_DIS
LIN {X -36.4895,Y 1.7874,Z 63,A 169.7011,B 24.8413,C -2.9062,E1 24.8401,E2 -446.5904} C_DIS
LIN {X -36.2743,Y 4.3451,Z 63,A 164.7254,B 24.8408,C -2.9104,E1 24.8415,E2 -441.5951} C_DIS
LIN {X -35.8639,Y 6.9622,Z 63,A 161.571,B 24.8384,C -2.9322,E1 24.843,E2 -438.4741} C_DIS
LIN {X -35.4123,Y 8.9817,Z 63,A 157.7147,B 24.8379,C -2.9368,E1 24.8455,E2 -434.6062} C_DIS
LIN {X -34.7814,Y 11.1783,Z 63,A 154.2251,B 24.8366,C -2.9485,E1 24.8483,E2 -431.1247} C_DIS
LIN {X -33.8506,Y 13.7416,Z 63,A 150.0602,B 24.8351,C -2.9623,E1 24.8525,E2 -426.9694} C_DIS
LIN {X -32.7891,Y 16.1116,Z 63,A 145.7026,B 24.834,C -2.9717,E1 24.8576,E2 -422.6104} C_DIS
LIN {X -31.8393,Y 17.9154,Z 63,A 143.0365,B 24.8325,C -2.9856,E1 24.8611,E2 -419.9634} C_DIS
LIN {X -30.724,Y 19.7669,Z 63,A 138.6521,B 24.8325,C -2.9858,E1 24.8677,E2 -415.5573} C_DIS
LIN {X -29.0467,Y 22.1588,Z 63,A 133.7463,B 24.8314,C -2.9949,E1 24.8759,E2 -410.6496} C_DIS
LIN {X -26.0618,Y 25.6024,Z 63,A 126.6875,B 24.8294,C -3.0131,E1 24.8892,E2 -403.6034} C_DIS
LIN {X -22.7831,Y 28.5596,Z 63,A 120.6682,B 24.8266,C -3.0371,E1 24.9018,E2 -397.6178} C_DIS
LIN {X -20.1605,Y 30.467,Z 63,A 114.7613,B 24.8264,C -3.0388,E1 24.9154,E2 -391.6949} C_DIS
LIN {X -17.8272,Y 31.8885,Z 63,A 111.2538,B 24.8246,C -3.0542,E1 24.9238,E2 -388.2136} C_DIS
LIN {X -15.848,Y 32.9171,Z 63,A 107.8041,B 24.824,C -3.0602,E1 24.9323,E2 -384.7691} C_DIS
LIN {X -13.9827,Y 33.7512,Z 63,A 104.5841,B 24.8234,C -3.0646,E1 24.9406,E2 -381.552} C_DIS
LIN {X -12.1916,Y 34.4393,Z 63,A 101.3908,B 24.8232,C -3.0665,E1 24.949,E2 -378.3565} C_DIS
LIN {X -10.5014,Y 34.9918,Z 63,A 98.7927,B 24.8226,C -3.0717,E1 24.9559,E2 -375.7663} C_DIS
LIN {X -8.9096,Y 35.4309,Z 63,A 95.7738,B 24.8229,C -3.0695,E1 24.964,E2 -372.7376} C_DIS
LIN {X -6.3545,Y 35.9766,Z 63,A 92.1097,B 24.8219,C -3.0776,E1 24.974,E2 -369.0888} C_DIS
LIN {X -4.3511,Y 36.2736,Z 63,A 88.5569,B 24.8222,C -3.0752,E1 24.9839,E2 -365.5277} C_DIS
LIN {X -2.3787,Y 36.456,Z 63,A 85.7868,B 24.8216,C -3.0805,E1 24.9916,E2 -362.7689} C_DIS
LIN {X -0.7382,Y 36.526,Z 63,A 83.1084,B 24.8216,C -3.08,E1 24.999,E2 -360.089} C_DIS
LIN {X 1.1293,Y 36.516,Z 63,A 80.0902,B 24.8217,C -3.0793,E1 25.0075,E2 -357.0697} C_DIS
LIN {X 3.38,Y 36.3768,Z 63,A 76.4361,B 24.8219,C -3.0778,E1 25.0177,E2 -353.4137} C_DIS
LIN {X 5.1545,Y 36.168,Z 63,A 73.8336,B 24.8217,C -3.0796,E1 25.0248,E2 -350.8176} C_DIS
LIN {X 7.0057,Y 35.8556,Z 63,A 70.9301,B 24.8217,C -3.079,E1 25.0328,E2 -347.9159} C_DIS
LIN {X 8.8224,Y 35.4521,Z 63,A 68.0464,B 24.8219,C -3.0779,E1 25.0406,E2 -345.0337} C_DIS
LIN {X 10.5992,Y 34.9628,Z 63,A 65.2618,B 24.8219,C -3.0773,E1 25.0481,E2 -342.2523} C_DIS
LIN {X 12.5041,Y 34.3269,Z 63,A 61.8213,B 24.8227,C -3.0709,E1 25.0572,E2 -338.8035} C_DIS
LIN {X 15.3754,Y 33.1405,Z 63,A 56.7067,B 24.8237,C -3.0626,E1 25.0703,E2 -333.6814} C_DIS
LIN {X 17.4759,Y 32.0825,Z 63,A 53.0418,B 24.8242,C -3.0581,E1 25.0794,E2 -330.0163} C_DIS
LIN {X 19.3829,Y 30.9677,Z 63,A 49.6836,B 24.8246,C -3.0545,E1 25.0874,E2 -326.66} C_DIS
LIN {X 21.0913,Y 29.8308,Z 63,A 46.8863,B 24.8246,C -3.055,E1 25.0938,E2 -323.8736} C_DIS
LIN {X 22.3096,Y 28.9305,Z 63,A 44.5969,B 24.8249,C -3.0522,E1 25.0989,E2 -321.5855} C_DIS
LIN {X 23.3607,Y 28.0885,Z 63,A 42.3902,B 24.8255,C -3.047,E1 25.1037,E2 -319.375} C_DIS
LIN {X 24.6706,Y 26.9454,Z 63,A 39.3712,B 24.8266,C -3.0376,E1 25.11,E2 -316.3457} C_DIS
LIN {X 26.1639,Y 25.4987,Z 63,A 36.4054,B 24.8269,C -3.035,E1 25.1158,E2 -313.3863} C_DIS
LIN {X 27.3962,Y 24.1696,Z 63,A 32.7955,B 24.8288,C -3.0178,E1 25.1226,E2 -309.7519} C_DIS
LIN {X 29.3019,Y 21.82,Z 63,A 28.9491,B 24.8286,C -3.0197,E1 25.1292,E2 -305.9279} C_DIS
LIN {X 30.5058,Y 20.1019,Z 63,A 25.3257,B 24.8301,C -3.0067,E1 25.1349,E2 -302.2916} C_DIS
LIN {X 31.6566,Y 18.236,Z 63,A 21.5433,B 24.8317,C -2.9927,E1 25.1403,E2 -298.4956} C_DIS
LIN {X 33.318,Y 14.9867,Z 63,A 16.9922,B 24.8315,C -2.9946,E1 25.1459,E2 -293.9733} C_DIS
LIN {X 33.9692,Y 13.4459,Z 63,A 13.5411,B 24.8337,C -2.9748,E1 25.1496,E2 -290.4942} C_DIS
LIN {X 34.7315,Y 11.3325,Z 63,A 10.2948,B 24.8344,C -2.9688,E1 25.1525,E2 -287.252} C_DIS
LIN {X 35.2641,Y 9.5467,Z 63,A 7.1611,B 24.8357,C -2.957,E1 25.1549,E2 -284.1083} C_DIS
LIN {X 35.8587,Y 6.9893,Z 63,A 3.153,B 24.8369,C -2.9462,E1 25.1573,E2 -280.098} C_DIS
LIN {X 36.1927,Y 4.9806,Z 63,A -0.0218,B 24.8379,C -2.9367,E1 25.1586,E2 -276.9193} C_DIS
LIN {X 36.4563,Y 2.3746,Z 63,A -4.0568,B 24.8392,C -2.9251,E1 25.1596,E2 -272.8808} C_DIS
LIN {X 36.5319,Y 0.3607,Z 63,A -8.0548,B 24.8417,C -2.9025,E1 25.1597,E2 -268.8531} C_DIS
LIN {X 36.4498,Y -2.4709,Z 63,A -12.4232,B 24.8431,C -2.8897,E1 25.159,E2 -264.4803} C_DIS
LIN {X 35.9707,Y -6.3883,Z 63,A -17.8117,B 24.8439,C -2.8825,E1 25.1569,E2 -259.1065} C_DIS
LIN {X 35.4596,Y -8.7936,Z 63,A -21.4192,B 24.8448,C -2.8743,E1 25.1547,E2 -255.5007} C_DIS
LIN {X 35.0218,Y -10.4002,Z 63,A -24.6441,B 24.8466,C -2.857,E1 25.1521,E2 -252.2532} C_DIS
LIN {X 33.7227,Y -14.0533,Z 63,A -30.0536,B 24.8475,C -2.8489,E1 25.1468,E2 -246.8546} C_DIS
LIN {X 32.7134,Y -16.2644,Z 63,A -34.2875,B 24.8494,C -2.8314,E1 25.1417,E2 -242.602} C_DIS
LIN {X 31.6874,Y -18.1824,Z 63,A -37.1024,B 24.8494,C -2.8306,E1 25.1379,E2 -239.8001} C_DIS
LIN {X 30.6966,Y -19.8095,Z 63,A -40.4507,B 24.8509,C -2.8169,E1 25.133,E2 -236.4362} C_DIS
LIN {X 29.5927,Y -21.4239,Z 63,A -43.2482,B 24.8514,C -2.8127,E1 25.1285,E2 -233.6424} C_DIS
LIN {X 28.4352,Y -22.9377,Z 63,A -46.3994,B 24.8525,C -2.8025,E1 25.123,E2 -230.4819} C_DIS
LIN {X 27.0247,Y -24.5842,Z 63,A -49.5075,B 24.8529,C -2.7983,E1 25.1173,E2 -227.3778} C_DIS
LIN {X 25.9903,Y -25.6748,Z 63,A -51.7439,B 24.8533,C -2.7944,E1 25.113,E2 -225.1418} C_DIS
LIN {X 25.026,Y -26.6156,Z 63,A -53.9017,B 24.8539,C -2.7888,E1 25.1086,E2 -222.9797} C_DIS
LIN {X 23.9638,Y -27.576,Z 63,A -56.1431,B 24.8544,C -2.7838,E1 25.1039,E2 -220.7354} C_DIS
LIN {X 22.9325,Y -28.4394,Z 63,A -58.5175,B 24.8553,C -2.7754,E1 25.0988,E2 -218.3502} C_DIS
LIN {X 21.187,Y -29.7625,Z 63,A -61.8481,B 24.8559,C -2.7699,E1 25.0913,E2 -215.0184} C_DIS
LIN {X 19.7727,Y -30.7203,Z 63,A -64.341,B 24.8561,C -2.7674,E1 25.0855,E2 -212.5278} C_DIS
LIN {X 18.0641,Y -31.7554,Z 63,A -67.9652,B 24.8574,C -2.755,E1 25.0767,E2 -208.8851} C_DIS
LIN {X 15.9654,Y -32.8605,Z 63,A -71.4001,B 24.8577,C -2.7529,E1 25.0682,E2 -205.4546} C_DIS
LIN {X 14.1365,Y -33.6874,Z 63,A -74.7182,B 24.8584,C -2.746,E1 25.0596,E2 -202.1281} C_DIS
LIN {X 12.4895,Y -34.3323,Z 63,A -77.2759,B 24.8584,C -2.7452,E1 25.053,E2 -199.5742} C_DIS
LIN {X 10.9073,Y -34.8673,Z 63,A -80.0952,B 24.859,C -2.7395,E1 25.0454,E2 -196.7465} C_DIS
LIN {X 8.5249,Y -35.5252,Z 63,A -83.8536,B 24.8593,C -2.7371,E1 25.0353,E2 -192.9883} C_DIS
LIN {X 6.3447,Y -35.9777,Z 63,A -87.1946,B 24.8593,C -2.7363,E1 25.0261,E2 -189.6491} C_DIS
LIN {X 4.4748,Y -36.259,Z 63,A -90.6988,B 24.8603,C -2.7274,E1 25.0164,E2 -186.1269} C_DIS
LIN {X 1.1721,Y -36.5145,Z 63,A -95.316,B 24.8598,C -2.7326,E1 25.0036,E2 -181.5237} C_DIS
LIN {X 1.1721,Y -36.5145,Z 63,A -95.316,B 24.8598,C -2.7326,E1 25.0036,E2 -181.5237} C_DIS
Enddeposition()
LIN {X 0.1757,Y -35.5825,Z 63,A -95.5143,B 24.8563,C -2.7656,E1 25.0032,E2 -181.4039} C_DIS
Startdeposition()
$VEL.CP = VEL_PRINT
LIN {X 2.189,Y -35.5166,Z 63,A -92.1914,B 24.8561,C -2.7678,E1 25.0125,E2 -184.731} C_DIS
LIN {X 4.2985,Y -35.3234,Z 63,A -89.107,B 24.8563,C -2.7655,E1 25.021,E2 -187.8079} C_DIS
LIN {X 5.486,Y -35.1581,Z 63,A -86.5985,B 24.8554,C -2.7743,E1 25.028,E2 -190.3349} C_DIS
LIN {X 8.5217,Y -34.5483,Z 63,A -81.1373,B 24.8543,C -2.7851,E1 25.0429,E2 -195.8145} C_DIS
LIN {X 12.3122,Y -33.3859,Z 63,A -75.6863,B 24.8548,C -2.7802,E1 25.0573,E2 -201.2433} C_DIS
LIN {X 14.1092,Y -32.6671,Z 63,A -71.4435,B 24.8527,C -2.8001,E1 25.0683,E2 -205.5234} C_DIS
LIN {X 17.8967,Y -30.7556,Z 63,A -64.9916,B 24.8521,C -2.8063,E1 25.0842,E2 -211.9714} C_DIS
LIN {X 19.7264,Y -29.6157,Z 63,A -62.2029,B 24.8524,C -2.8032,E1 25.0906,E2 -214.7436} C_DIS
LIN {X 21.3585,Y -28.4607,Z 63,A -58.9719,B 24.8517,C -2.8099,E1 25.0979,E2 -217.9791} C_DIS
LIN {X 22.7823,Y -27.3343,Z 63,A -55.9761,B 24.8509,C -2.8172,E1 25.1044,E2 -220.981} C_DIS
LIN {X 24.3695,Y -25.9292,Z 63,A -52.6483,B 24.8502,C -2.8238,E1 25.1113,E2 -224.3108} C_DIS
LIN {X 26.1257,Y -24.1591,Z 63,A -48.3566,B 24.8487,C -2.8375,E1 25.1196,E2 -228.6165} C_DIS
LIN {X 27.7587,Y -22.2638,Z 63,A -44.9374,B 24.8487,C -2.8388,E1 25.1257,E2 -232.023} C_DIS
LIN {X 28.7386,Y -20.9822,Z 63,A -41.5806,B 24.8466,C -2.857,E1 25.1313,E2 -235.4068} C_DIS
LIN {X 30.6199,Y -18.1278,Z 63,A -37.0462,B 24.8466,C -2.8576,E1 25.1381,E2 -239.9199} C_DIS
LIN {X 31.3632,Y -16.8099,Z 63,A -33.8896,B 24.8447,C -2.8754,E1 25.1424,E2 -243.1021} C_DIS
LIN {X 32.6497,Y -14.1491,Z 63,A -29.5241,B 24.8438,C -2.8834,E1 25.1475,E2 -247.4629} C_DIS
LIN {X 33.407,Y -12.2543,Z 63,A -25.9548,B 24.8422,C -2.8976,E1 25.1511,E2 -251.046} C_DIS
LIN {X 34.0896,Y -10.2028,Z 63,A -22.638,B 24.8414,C -2.9057,E1 25.1538,E2 -254.3631} C_DIS
LIN {X 34.6846,Y -7.9483,Z 63,A -19.085,B 24.8404,C -2.9142,E1 25.1562,E2 -257.9158} C_DIS
LIN {X 35.041,Y -6.1914,Z 63,A -15.6872,B 24.8386,C -2.9311,E1 25.1579,E2 -261.3336} C_DIS
LIN {X 35.4685,Y -2.8594,Z 63,A -10.9059,B 24.8377,C -2.9384,E1 25.1594,E2 -266.1039} C_DIS
LIN {X 35.5836,Y 0.0716,Z 63,A -6.6621,B 24.8369,C -2.9459,E1 25.1598,E2 -270.3402} C_DIS
LIN {X 35.5482,Y 1.5883,Z 63,A -3.602,B 24.835,C -2.9629,E1 25.1595,E2 -273.4224} C_DIS
LIN {X 35.367,Y 3.9192,Z 63,A -0.0876,B 24.8341,C -2.9708,E1 25.1586,E2 -276.9346} C_DIS
LIN {X 35.1462,Y 5.5637,Z 63,A 2.9584,B 24.8326,C -2.9846,E1 25.1573,E2 -279.9955} C_DIS
LIN {X 34.696,Y 7.899,Z 63,A 6.9365,B 24.831,C -2.9985,E1 25.155,E2 -283.9832} C_DIS
LIN {X 34.154,Y 9.986,Z 63,A 9.7154,B 24.831,C -2.9983,E1 25.153,E2 -286.7457} C_DIS
LIN {X 33.7323,Y 11.3281,Z 63,A 12.0409,B 24.8302,C -3.0058,E1 25.1509,E2 -289.0758} C_DIS
LIN {X 33.2613,Y 12.6445,Z 63,A 14.2162,B 24.8296,C -3.0111,E1 25.1488,E2 -291.2515} C_DIS
LIN {X 32.5471,Y 14.3844,Z 63,A 17.6139,B 24.828,C -3.0251,E1 25.1451,E2 -294.6636} C_DIS
LIN {X 31.4162,Y 16.7089,Z 63,A 21.5144,B 24.8271,C -3.0324,E1 25.1402,E2 -298.5609} C_DIS
LIN {X 30.5525,Y 18.2418,Z 63,A 24.3142,B 24.8264,C -3.0393,E1 25.1363,E2 -301.3626} C_DIS
LIN {X 29.6338,Y 19.6989,Z 63,A 27.2954,B 24.8252,C -3.0493,E1 25.1317,E2 -304.3525} C_DIS
LIN {X 28.3112,Y 21.5571,Z 63,A 30.9902,B 24.8242,C -3.0584,E1 25.1256,E2 -308.0512} C_DIS
LIN {X 26.6322,Y 23.5998,Z 63,A 35.1789,B 24.8232,C -3.067,E1 25.118,E2 -312.2411} C_DIS
LIN {X 25.0703,Y 25.2523,Z 63,A 38.7561,B 24.8224,C -3.0735,E1 25.111,E2 -315.8184} C_DIS
LIN {X 23.6476,Y 26.589,Z 63,A 42.1171,B 24.8213,C -3.0827,E1 25.1041,E2 -319.1878} C_DIS
LIN {X 21.6319,Y 28.2536,Z 63,A 45.7895,B 24.8213,C -3.0829,E1 25.0961,E2 -322.8467} C_DIS
LIN {X 20.4957,Y 29.0888,Z 63,A 47.9786,B 24.821,C -3.0855,E1 25.0911,E2 -325.0344} C_DIS
LIN {X 18.693,Y 30.2787,Z 63,A 51.8183,B 24.8198,C -3.0958,E1 25.0821,E2 -328.8859} C_DIS
Enddeposition()
END
